QRS_NEXT_CUT()
PTP {E1 28256.982,E2 28256.982}
PTP {X 0,Y 607.876,A -85,B 0,C 180,E1 28256.982,E2 28256.982,E3 0,E4 0,E5 0,E6 0}
QRS_SPEED_INIT()
LIN {X 0,Y 607.876,Z 951,A -85,B 0,C 180,E1 28256.982,E2 28256.982,E3 0,E4 0,E5 0,E6 0} C_VEL
LIN {X 0,Y 607.876,Z 233.398,A -85,B 0,C 180,E1 28256.982,E2 28256.982} C_VEL
LIN {X 0,Y 607.876,Z 225.322,A -85,B 0,C 180,E1 28256.982,E2 28256.982} C_VEL
LIN {X 0,Y 607.869,Z 223.322,A -85,B 0,C 180,E1 28256.793,E2 28256.793} C_VEL
LIN {X 0,Y 607.913,Z 223.325,A -85,B 0,C 180,E1 28253.769,E2 28253.769} C_VEL
LIN {X 0,Y 607.873,Z 223.321,A -85,B 0,C 180,E1 28250.629,E2 28250.629} C_VEL
LIN {X 0,Y 607.911,Z 223.323,A -85,B 0,C 180,E1 28247.558,E2 28247.558} C_VEL
LIN {X 0,Y 607.877,Z 223.322,A -85,B 0,C 180,E1 28244.449,E2 28244.449} C_VEL
LIN {X 0,Y 607.908,Z 223.321,A -85,B 0,C 180,E1 28241.331,E2 28241.331} C_VEL
LIN {X 0,Y 607.881,Z 223.322,A -85,B 0,C 180,E1 28238.28,E2 28238.28} C_VEL
LIN {X 0,Y 607.906,Z 223.322,A -85,B 0,C 180,E1 28235.203,E2 28235.203} C_VEL
LIN {X 0,Y 607.886,Z 223.323,A -85,B 0,C 180,E1 28232.039,E2 28232.039} C_VEL
LIN {X 0,Y 607.905,Z 223.32,A -85,B 0,C 180,E1 28228.906,E2 28228.906} C_VEL
LIN {X 0,Y 607.894,Z 223.324,A -85,B 0,C 180,E1 28225.771,E2 28225.771} C_VEL
LIN {X 0,Y 607.909,Z 223.317,A -85,B 0,C 180,E1 28222.516,E2 28222.516} C_VEL
LIN {X 0,Y 607.913,Z 223.326,A -85,B 0,C 180,E1 28219.236,E2 28219.236} C_VEL
LIN {X 0,Y 607.898,Z 223.319,A -85,B 0,C 180,E1 28215.954,E2 28215.954} C_VEL
LIN {X 0,Y 607.896,Z 223.322,A -85,B 0,C 180,E1 28212.789,E2 28212.789} C_VEL
LIN {X 0,Y 607.898,Z 223.321,A -85,B 0,C 180,E1 28209.656,E2 28209.656} C_VEL
LIN {X 0,Y 607.891,Z 223.321,A -85,B 0,C 180,E1 28206.543,E2 28206.543} C_VEL
LIN {X 0,Y 607.902,Z 223.322,A -85,B 0,C 180,E1 28203.436,E2 28203.436} C_VEL
LIN {X 0,Y 607.889,Z 223.32,A -85,B 0,C 180,E1 28200.287,E2 28200.287} C_VEL
LIN {X 0,Y 607.91,Z 223.325,A -85,B 0,C 180,E1 28197.104,E2 28197.104} C_VEL
LIN {X 0,Y 607.899,Z 223.318,A -85,B 0,C 180,E1 28193.868,E2 28193.868} C_VEL
LIN {X 0,Y 607.897,Z 223.326,A -85,B 0,C 180,E1 28190.609,E2 28190.609} C_VEL
LIN {X 0,Y 607.916,Z 223.317,A -85,B 0,C 180,E1 28187.419,E2 28187.419} C_VEL
LIN {X 0,Y 607.881,Z 223.324,A -85,B 0,C 180,E1 28184.285,E2 28184.285} C_VEL
LIN {X 0,Y 607.914,Z 223.318,A -85,B 0,C 180,E1 28181.192,E2 28181.192} C_VEL
LIN {X 0,Y 607.873,Z 223.326,A -85,B 0,C 180,E1 28178.035,E2 28178.035} C_VEL
LIN {X 0,Y 607.913,Z 223.532,A -85,B 0,C 180,E1 28176.802,E2 28176.802} C_VEL
LIN {X 0,Y 607.916,Z 225.924,A -85,B 0,C 180,E1 28176.612,E2 28176.612} C_VEL
LIN {X 0,Y 607.89,Z 279.402,A -85,B 0,C 180,E1 28173.632,E2 28173.632} C_VEL
LIN {X 0,Y 607.913,Z 336.91,A -85,B 0,C 180,E1 28170.519,E2 28170.519} C_VEL
LIN {X 0,Y 607.902,Z 395.097,A -85,B 0,C 180,E1 28167.456,E2 28167.456} C_VEL
LIN {X 0,Y 607.896,Z 417.723,A -85,B 0,C 180,E1 28166.3,E2 28166.3} C_VEL
LIN {X 0,Y 607.917,Z 627.491,A -85,B 0,C 180,E1 28163.674,E2 28163.674} C_VEL
LIN {X 0,Y 607.913,Z 646.173,A -85,B 0,C 180,E1 28163.271,E2 28163.271} C_VEL
LIN {X 0,Y 607.918,Z 664.898,A -85,B 0,C 180,E1 28162.681,E2 28162.681} C_VEL
LIN {X 0,Y 607.911,Z 682.608,A -85,B 0,C 180,E1 28161.94,E2 28161.94} C_VEL
LIN {X 0,Y 607.919,Z 700.049,A -85,B 0,C 180,E1 28161.012,E2 28161.012} C_VEL
LIN {X 0,Y 607.919,Z 716.108,A -85,B 0,C 180,E1 28159.961,E2 28159.961} C_VEL
LIN {X 0,Y 607.915,Z 731.242,A -85,B 0,C 180,E1 28158.762,E2 28158.762} C_VEL
LIN {X 0,Y 607.916,Z 744.939,A -85,B 0,C 180,E1 28157.462,E2 28157.462} C_VEL
LIN {X 0,Y 607.919,Z 757.696,A -85,B 0,C 180,E1 28156.01,E2 28156.01} C_VEL
LIN {X 0,Y 607.915,Z 769.022,A -85,B 0,C 180,E1 28154.45,E2 28154.45} C_VEL
LIN {X 0,Y 607.913,Z 778.456,A -85,B 0,C 180,E1 28152.858,E2 28152.858} C_VEL
LIN {X 0,Y 607.908,Z 786.332,A -85,B 0,C 180,E1 28151.195,E2 28151.195} C_VEL
LIN {X 0,Y 607.913,Z 792.505,A -85,B 0,C 180,E1 28149.494,E2 28149.494} C_VEL
LIN {X 0,Y 607.919,Z 796.976,A -85,B 0,C 180,E1 28147.774,E2 28147.774} C_VEL
LIN {X 0,Y 607.908,Z 799.783,A -85,B 0,C 180,E1 28146.032,E2 28146.032} C_VEL
LIN {X 0,Y 607.912,Z 800.933,A -85,B 0,C 180,E1 28144.266,E2 28144.266} C_VEL
LIN {X 0,Y 607.912,Z 800.367,A -85,B 0,C 180,E1 28142.474,E2 28142.474} C_VEL
LIN {X 0,Y 607.912,Z 798.18,A -85,B 0,C 180,E1 28140.76,E2 28140.76} C_VEL
LIN {X 0,Y 607.914,Z 794.265,A -85,B 0,C 180,E1 28139.017,E2 28139.017} C_VEL
LIN {X 0,Y 607.908,Z 788.856,A -85,B 0,C 180,E1 28137.353,E2 28137.353} C_VEL
LIN {X 0,Y 607.916,Z 781.522,A -85,B 0,C 180,E1 28135.654,E2 28135.654} C_VEL
LIN {X 0,Y 607.913,Z 772.553,A -85,B 0,C 180,E1 28134.018,E2 28134.018} C_VEL
LIN {X 0,Y 607.914,Z 762.445,A -85,B 0,C 180,E1 28132.517,E2 28132.517} C_VEL
LIN {X 0,Y 607.915,Z 750.725,A -85,B 0,C 180,E1 28131.073,E2 28131.073} C_VEL
LIN {X 0,Y 607.914,Z 737.718,A -85,B 0,C 180,E1 28129.733,E2 28129.733} C_VEL
LIN {X 0,Y 607.917,Z 723.253,A -85,B 0,C 180,E1 28128.486,E2 28128.486} C_VEL
LIN {X 0,Y 607.917,Z 707.272,A -85,B 0,C 180,E1 28127.343,E2 28127.343} C_VEL
LIN {X 0,Y 607.896,Z 690.448,A -85,B 0,C 180,E1 28126.36,E2 28126.36} C_VEL
LIN {X 0,Y 607.915,Z 672.447,A -85,B 0,C 180,E1 28125.522,E2 28125.522} C_VEL
LIN {X 0,Y 607.915,Z 654.423,A -85,B 0,C 180,E1 28124.876,E2 28124.876} C_VEL
LIN {X 0,Y 607.913,Z 636.158,A -85,B 0,C 180,E1 28124.401,E2 28124.401} C_VEL
LIN {X 0,Y 607.919,Z 616.8,A -85,B 0,C 180,E1 28124.083,E2 28124.083} C_VEL
LIN {X 0,Y 607.917,Z 417.224,A -85,B 0,C 180,E1 28121.598,E2 28121.598} C_VEL
LIN {X 0,Y 607.897,Z 358.995,A -85,B 0,C 180,E1 28118.562,E2 28118.562} C_VEL
LIN {X 0,Y 607.915,Z 298.763,A -85,B 0,C 180,E1 28115.337,E2 28115.337} C_VEL
LIN {X 0,Y 607.915,Z 242.721,A -85,B 0,C 180,E1 28112.245,E2 28112.245} C_VEL
LIN {X 0,Y 607.894,Z 223.784,A -85,B 0,C 180,E1 28111.15,E2 28111.15} C_VEL
LIN {X 0,Y 607.854,Z 223.332,A -85,B 0,C 180,E1 28110.839,E2 28110.839} C_VEL
LIN {X 0,Y 607.831,Z 223.328,A -85,B 0,C 180,E1 28108.063,E2 28108.063} C_VEL
LIN {X 0,Y 607.896,Z 223.327,A -85,B 0,C 180,E1 28105.005,E2 28105.005} C_VEL
LIN {X 0,Y 607.827,Z 223.327,A -85,B 0,C 180,E1 28102.129,E2 28102.129} C_VEL
LIN {X 0,Y 607.89,Z 223.327,A -85,B 0,C 180,E1 28099.205,E2 28099.205} C_VEL
LIN {X 0,Y 607.83,Z 223.327,A -85,B 0,C 180,E1 28096.131,E2 28096.131} C_VEL
LIN {X 0,Y 607.845,Z 223.327,A -85,B 0,C 180,E1 28093.41,E2 28093.41} C_VEL
LIN {X 0,Y 607.839,Z 223.327,A -85,B 0,C 180,E1 28090.137,E2 28090.137} C_VEL
LIN {X 0,Y 607.83,Z 223.327,A -85,B 0,C 180,E1 28087.466,E2 28087.466} C_VEL
LIN {X 0,Y 607.877,Z 223.327,A -85,B 0,C 180,E1 28084.339,E2 28084.339} C_VEL
LIN {X 0,Y 607.824,Z 223.327,A -85,B 0,C 180,E1 28081.508,E2 28081.508} C_VEL
LIN {X 0,Y 607.913,Z 223.327,A -85,B 0,C 180,E1 28078.492,E2 28078.492} C_VEL
LIN {X 0,Y 607.824,Z 223.327,A -85,B 0,C 180,E1 28075.471,E2 28075.471} C_VEL
LIN {X 0,Y 607.845,Z 223.327,A -85,B 0,C 180,E1 28072.818,E2 28072.818} C_VEL
LIN {X 0,Y 607.836,Z 223.328,A -85,B 0,C 180,E1 28069.575,E2 28069.575} C_VEL
LIN {X 0,Y 607.83,Z 223.327,A -85,B 0,C 180,E1 28066.853,E2 28066.853} C_VEL
LIN {X 0,Y 607.859,Z 223.327,A -85,B 0,C 180,E1 28063.663,E2 28063.663} C_VEL
LIN {X 0,Y 607.823,Z 223.327,A -85,B 0,C 180,E1 28060.892,E2 28060.892} C_VEL
LIN {X 0,Y 607.905,Z 223.327,A -85,B 0,C 180,E1 28057.815,E2 28057.815} C_VEL
LIN {X 0,Y 607.824,Z 223.327,A -85,B 0,C 180,E1 28054.887,E2 28054.887} C_VEL
LIN {X 0,Y 607.871,Z 223.328,A -85,B 0,C 180,E1 28052.038,E2 28052.038} C_VEL
LIN {X 0,Y 607.83,Z 223.327,A -85,B 0,C 180,E1 28048.901,E2 28048.901} C_VEL
LIN {X 0,Y 607.837,Z 223.327,A -85,B 0,C 180,E1 28046.221,E2 28046.221} C_VEL
LIN {X 0,Y 607.839,Z 223.327,A -85,B 0,C 180,E1 28042.865,E2 28042.865} C_VEL
LIN {X 0,Y 607.835,Z 223.328,A -85,B 0,C 180,E1 28040.094,E2 28040.094} C_VEL
LIN {X 0,Y 607.86,Z 223.326,A -85,B 0,C 180,E1 28036.912,E2 28036.912} C_VEL
LIN {X 0,Y 607.829,Z 223.327,A -85,B 0,C 180,E1 28034.091,E2 28034.091} C_VEL
LIN {X 0,Y 607.873,Z 223.59,A -85,B 0,C 180,E1 28031.49,E2 28031.49} C_VEL
LIN {X 0,Y 607.887,Z 224.472,A -85,B 0,C 180,E1 28031.391,E2 28031.391} C_VEL
LIN {X 0,Y 607.917,Z 283.251,A -85,B 0,C 180,E1 28028.68,E2 28028.68} C_VEL
LIN {X 0,Y 607.918,Z 312.017,A -85,B 0,C 180,E1 28027.401,E2 28027.401} C_VEL
LIN {X 0,Y 607.918,Z 518.654,A -85,B 0,C 180,E1 28024.442,E2 28024.442} C_VEL
LIN {X 0,Y 607.912,Z 661.034,A -85,B 0,C 180,E1 28022.442,E2 28022.442} C_VEL
LIN {X 0,Y 607.919,Z 684.142,A -85,B 0,C 180,E1 28021.955,E2 28021.955} C_VEL
LIN {X 0,Y 607.916,Z 703.574,A -85,B 0,C 180,E1 28021.393,E2 28021.393} C_VEL
LIN {X 0,Y 607.913,Z 724.964,A -85,B 0,C 180,E1 28020.626,E2 28020.626} C_VEL
LIN {X 0,Y 607.919,Z 745.116,A -85,B 0,C 180,E1 28019.725,E2 28019.725} C_VEL
LIN {X 0,Y 607.916,Z 765.788,A -85,B 0,C 180,E1 28018.647,E2 28018.647} C_VEL
LIN {X 0,Y 607.917,Z 785.585,A -85,B 0,C 180,E1 28017.419,E2 28017.419} C_VEL
LIN {X 0,Y 607.915,Z 804.976,A -85,B 0,C 180,E1 28016.048,E2 28016.048} C_VEL
LIN {X 0,Y 607.912,Z 823.181,A -85,B 0,C 180,E1 28014.558,E2 28014.558} C_VEL
LIN {X 0,Y 607.909,Z 841.611,A -85,B 0,C 180,E1 28012.839,E2 28012.839} C_VEL
LIN {X 0,Y 607.905,Z 857.887,A -85,B 0,C 180,E1 28011.111,E2 28011.111} C_VEL
LIN {X 0,Y 607.906,Z 873.086,A -85,B 0,C 180,E1 28009.25,E2 28009.25} C_VEL
LIN {X 0,Y 607.907,Z 887.525,A -85,B 0,C 180,E1 28007.22,E2 28007.22} C_VEL
LIN {X 0,Y 607.916,Z 899.042,A -85,B 0,C 180,E1 28005.354,E2 28005.354} C_VEL
LIN {X 0,Y 607.917,Z 909.76,A -85,B 0,C 180,E1 28003.311,E2 28003.311} C_VEL
LIN {X 0,Y 607.916,Z 918.789,A -85,B 0,C 180,E1 28001.286,E2 28001.286} C_VEL
LIN {X 0,Y 607.919,Z 926.346,A -85,B 0,C 180,E1 27999.179,E2 27999.179} C_VEL
LIN {X 0,Y 607.913,Z 932.358,A -85,B 0,C 180,E1 27997.085,E2 27997.085} C_VEL
LIN {X 0,Y 607.908,Z 936.64,A -85,B 0,C 180,E1 27995,E2 27995} C_VEL
LIN {X 0,Y 607.915,Z 939.406,A -85,B 0,C 180,E1 27993.016,E2 27993.016} C_VEL
LIN {X 0,Y 607.906,Z 940.806,A -85,B 0,C 180,E1 27990.847,E2 27990.847} C_VEL
LIN {X 0,Y 607.918,Z 940.738,A -85,B 0,C 180,E1 27988.868,E2 27988.868} C_VEL
LIN {X 0,Y 607.909,Z 939.065,A -85,B 0,C 180,E1 27986.699,E2 27986.699} C_VEL
LIN {X 0,Y 607.909,Z 936.159,A -85,B 0,C 180,E1 27984.714,E2 27984.714} C_VEL
LIN {X 0,Y 607.913,Z 931.332,A -85,B 0,C 180,E1 27982.533,E2 27982.533} C_VEL
LIN {X 0,Y 607.91,Z 925.729,A -85,B 0,C 180,E1 27980.628,E2 27980.628} C_VEL
LIN {X 0,Y 607.91,Z 917.553,A -85,B 0,C 180,E1 27978.424,E2 27978.424} C_VEL
LIN {X 0,Y 607.918,Z 909.286,A -85,B 0,C 180,E1 27976.59,E2 27976.59} C_VEL
LIN {X 0,Y 607.912,Z 897.869,A -85,B 0,C 180,E1 27974.448,E2 27974.448} C_VEL
LIN {X 0,Y 607.919,Z 886.225,A -85,B 0,C 180,E1 27972.581,E2 27972.581} C_VEL
LIN {X 0,Y 607.915,Z 871.875,A -85,B 0,C 180,E1 27970.595,E2 27970.595} C_VEL
LIN {X 0,Y 607.91,Z 856.976,A -85,B 0,C 180,E1 27968.786,E2 27968.786} C_VEL
LIN {X 0,Y 607.909,Z 840.575,A -85,B 0,C 180,E1 27967.057,E2 27967.057} C_VEL
LIN {X 0,Y 607.917,Z 822.199,A -85,B 0,C 180,E1 27965.358,E2 27965.358} C_VEL
LIN {X 0,Y 607.914,Z 803.588,A -85,B 0,C 180,E1 27963.845,E2 27963.845} C_VEL
LIN {X 0,Y 607.918,Z 784.749,A -85,B 0,C 180,E1 27962.525,E2 27962.525} C_VEL
LIN {X 0,Y 607.917,Z 764.763,A -85,B 0,C 180,E1 27961.297,E2 27961.297} C_VEL
LIN {X 0,Y 607.919,Z 745.116,A -85,B 0,C 180,E1 27960.275,E2 27960.275} C_VEL
LIN {X 0,Y 607.914,Z 724.087,A -85,B 0,C 180,E1 27959.339,E2 27959.339} C_VEL
LIN {X 0,Y 607.916,Z 703.574,A -85,B 0,C 180,E1 27958.607,E2 27958.607} C_VEL
LIN {X 0,Y 607.919,Z 684.1,A -85,B 0,C 180,E1 27958.044,E2 27958.044} C_VEL
LIN {X 0,Y 607.911,Z 662.086,A -85,B 0,C 180,E1 27957.575,E2 27957.575} C_VEL
LIN {X 0,Y 607.908,Z 431.434,A -85,B 0,C 180,E1 27954.325,E2 27954.325} C_VEL
LIN {X 0,Y 607.918,Z 311.433,A -85,B 0,C 180,E1 27952.578,E2 27952.578} C_VEL
LIN {X 0,Y 607.918,Z 247.749,A -85,B 0,C 180,E1 27949.699,E2 27949.699} C_VEL
LIN {X 0,Y 607.88,Z 223.942,A -85,B 0,C 180,E1 27948.565,E2 27948.565} C_VEL
LIN {X 0,Y 607.855,Z 223.344,A -85,B 0,C 180,E1 27948.352,E2 27948.352} C_VEL
LIN {X 0,Y 607.826,Z 223.327,A -85,B 0,C 180,E1 27945.643,E2 27945.643} C_VEL
LIN {X 0,Y 607.893,Z 223.327,A -85,B 0,C 180,E1 27942.533,E2 27942.533} C_VEL
LIN {X 0,Y 607.828,Z 223.327,A -85,B 0,C 180,E1 27939.659,E2 27939.659} C_VEL
LIN {X 0,Y 607.911,Z 223.328,A -85,B 0,C 180,E1 27936.617,E2 27936.617} C_VEL
LIN {X 0,Y 607.834,Z 223.326,A -85,B 0,C 180,E1 27933.553,E2 27933.553} C_VEL
LIN {X 0,Y 607.892,Z 223.327,A -85,B 0,C 180,E1 27930.656,E2 27930.656} C_VEL
LIN {X 0,Y 607.843,Z 223.325,A -85,B 0,C 180,E1 27927.531,E2 27927.531} C_VEL
LIN {X 0,Y 607.891,Z 223.327,A -85,B 0,C 180,E1 27924.591,E2 27924.591} C_VEL
LIN {X 0,Y 607.85,Z 223.324,A -85,B 0,C 180,E1 27921.418,E2 27921.418} C_VEL
LIN {X 0,Y 607.9,Z 223.327,A -85,B 0,C 180,E1 27918.409,E2 27918.409} C_VEL
LIN {X 0,Y 607.855,Z 223.323,A -85,B 0,C 180,E1 27915.259,E2 27915.259} C_VEL
LIN {X 0,Y 607.905,Z 223.328,A -85,B 0,C 180,E1 27912.25,E2 27912.25} C_VEL
LIN {X 0,Y 607.859,Z 223.323,A -85,B 0,C 180,E1 27909.086,E2 27909.086} C_VEL
LIN {X 0,Y 607.918,Z 223.326,A -85,B 0,C 180,E1 27906.043,E2 27906.043} C_VEL
LIN {X 0,Y 607.864,Z 223.323,A -85,B 0,C 180,E1 27902.923,E2 27902.923} C_VEL
LIN {X 0,Y 607.916,Z 223.326,A -85,B 0,C 180,E1 27899.906,E2 27899.906} C_VEL
LIN {X 0,Y 607.869,Z 223.322,A -85,B 0,C 180,E1 27896.793,E2 27896.793} C_VEL
LIN {X 0,Y 606.876,Z 223.455,A -85,B 0,C 180,E1 27896.067,E2 27896.067} C_VEL
LIN {X 0,Y 600.494,Z 224.252,A -85,B 0,C 180,E1 27894.03,E2 27894.03} C_VEL
LIN {X 0,Y 599.974,Z 224.31,A -85,B 0,C 180,E1 27893.5,E2 27893.5} C_VEL
LIN {X 0,Y 599.935,Z 224.311,A -85,B 0,C 180,E1 27890.407,E2 27890.407} C_VEL
LIN {X 0,Y 599.973,Z 224.307,A -85,B 0,C 180,E1 27887.195,E2 27887.195} C_VEL
LIN {X 0,Y 599.958,Z 224.314,A -85,B 0,C 180,E1 27883.94,E2 27883.94} C_VEL
LIN {X 0,Y 599.95,Z 224.307,A -85,B 0,C 180,E1 27880.611,E2 27880.611} C_VEL
LIN {X 0,Y 599.971,Z 224.313,A -85,B 0,C 180,E1 27877.406,E2 27877.406} C_VEL
LIN {X 0,Y 599.945,Z 224.31,A -85,B 0,C 180,E1 27874.217,E2 27874.217} C_VEL
LIN {X 0,Y 599.966,Z 224.308,A -85,B 0,C 180,E1 27871.037,E2 27871.037} C_VEL
LIN {X 0,Y 599.953,Z 224.313,A -85,B 0,C 180,E1 27867.846,E2 27867.846} C_VEL
LIN {X 0,Y 599.97,Z 224.306,A -85,B 0,C 180,E1 27864.581,E2 27864.581} C_VEL
LIN {X 0,Y 599.973,Z 224.314,A -85,B 0,C 180,E1 27861.254,E2 27861.254} C_VEL
LIN {X 0,Y 599.959,Z 224.308,A -85,B 0,C 180,E1 27858.012,E2 27858.012} C_VEL
LIN {X 0,Y 599.958,Z 224.311,A -85,B 0,C 180,E1 27854.826,E2 27854.826} C_VEL
LIN {X 0,Y 599.959,Z 224.31,A -85,B 0,C 180,E1 27851.679,E2 27851.679} C_VEL
LIN {X 0,Y 599.954,Z 224.31,A -85,B 0,C 180,E1 27848.558,E2 27848.558} C_VEL
LIN {X 0,Y 599.964,Z 224.312,A -85,B 0,C 180,E1 27845.421,E2 27845.421} C_VEL
LIN {X 0,Y 599.955,Z 224.308,A -85,B 0,C 180,E1 27842.229,E2 27842.229} C_VEL
LIN {X 0,Y 599.971,Z 224.316,A -85,B 0,C 180,E1 27838.966,E2 27838.966} C_VEL
LIN {X 0,Y 599.976,Z 224.306,A -85,B 0,C 180,E1 27835.636,E2 27835.636} C_VEL
LIN {X 0,Y 599.945,Z 224.308,A -85,B 0,C 180,E1 27832.437,E2 27832.437} C_VEL
LIN {X 0,Y 599.97,Z 224.31,A -85,B 0,C 180,E1 27829.268,E2 27829.268} C_VEL
LIN {X 0,Y 599.939,Z 224.31,A -85,B 0,C 180,E1 27826.161,E2 27826.161} C_VEL
LIN {X 0,Y 599.971,Z 224.312,A -85,B 0,C 180,E1 27823.002,E2 27823.002} C_VEL
LIN {X 0,Y 599.935,Z 224.312,A -85,B 0,C 180,E1 27819.885,E2 27819.885} C_VEL
LIN {X 0,Y 599.992,Z 224.477,A -85,B 0,C 180,E1 27817.277,E2 27817.277} C_VEL
LIN {X 0,Y 600.467,Z 226.248,A -85,B 0,C 180,E1 27817.066,E2 27817.066} C_VEL
LIN {X 0,Y 600.943,Z 227.973,A -85,B 0,C 180,E1 27816.929,E2 27816.929} C_VEL
LIN {X 0,Y 600.723,Z 280.481,A -85,B 0,C 180,E1 27813.962,E2 27813.962} C_VEL
LIN {X 0,Y 600.585,Z 337.974,A -85,B 0,C 180,E1 27810.812,E2 27810.812} C_VEL
LIN {X 0,Y 600.431,Z 396.149,A -85,B 0,C 180,E1 27807.711,E2 27807.711} C_VEL
LIN {X 0,Y 600.462,Z 418.081,A -85,B 0,C 180,E1 27806.585,E2 27806.585} C_VEL
LIN {X 0,Y 600.377,Z 628.417,A -85,B 0,C 180,E1 27803.916,E2 27803.916} C_VEL
LIN {X 0,Y 600.334,Z 647.321,A -85,B 0,C 180,E1 27803.492,E2 27803.492} C_VEL
LIN {X 0,Y 600.295,Z 665.08,A -85,B 0,C 180,E1 27802.921,E2 27802.921} C_VEL
LIN {X 0,Y 600.227,Z 683.158,A -85,B 0,C 180,E1 27802.15,E2 27802.15} C_VEL
LIN {X 0,Y 600.177,Z 700.139,A -85,B 0,C 180,E1 27801.233,E2 27801.233} C_VEL
LIN {X 0,Y 600.119,Z 716.195,A -85,B 0,C 180,E1 27800.168,E2 27800.168} C_VEL
LIN {X 0,Y 600.064,Z 731.534,A -85,B 0,C 180,E1 27798.934,E2 27798.934} C_VEL
LIN {X 0,Y 600.018,Z 745.821,A -85,B 0,C 180,E1 27797.55,E2 27797.55} C_VEL
LIN {X 0,Y 599.984,Z 758.138,A -85,B 0,C 180,E1 27796.116,E2 27796.116} C_VEL
LIN {X 0,Y 599.953,Z 768.734,A -85,B 0,C 180,E1 27794.635,E2 27794.635} C_VEL
LIN {X 0,Y 599.934,Z 778.102,A -85,B 0,C 180,E1 27793.044,E2 27793.044} C_VEL
LIN {X 0,Y 599.92,Z 786.135,A -85,B 0,C 180,E1 27791.339,E2 27791.339} C_VEL
LIN {X 0,Y 599.915,Z 792.355,A -85,B 0,C 180,E1 27789.616,E2 27789.616} C_VEL
LIN {X 0,Y 599.915,Z 796.872,A -85,B 0,C 180,E1 27787.874,E2 27787.874} C_VEL
LIN {X 0,Y 599.911,Z 799.725,A -85,B 0,C 180,E1 27786.11,E2 27786.11} C_VEL
LIN {X 0,Y 599.913,Z 800.921,A -85,B 0,C 180,E1 27784.322,E2 27784.322} C_VEL
LIN {X 0,Y 599.912,Z 800.404,A -85,B 0,C 180,E1 27782.507,E2 27782.507} C_VEL
LIN {X 0,Y 599.913,Z 798.267,A -85,B 0,C 180,E1 27780.77,E2 27780.77} C_VEL
LIN {X 0,Y 599.916,Z 794.405,A -85,B 0,C 180,E1 27779.004,E2 27779.004} C_VEL
LIN {X 0,Y 599.915,Z 789.04,A -85,B 0,C 180,E1 27777.315,E2 27777.315} C_VEL
LIN {X 0,Y 599.93,Z 781.726,A -85,B 0,C 180,E1 27775.585,E2 27775.585} C_VEL
LIN {X 0,Y 599.944,Z 772.815,A -85,B 0,C 180,E1 27773.928,E2 27773.928} C_VEL
LIN {X 0,Y 599.967,Z 762.233,A -85,B 0,C 180,E1 27772.334,E2 27772.334} C_VEL
LIN {X 0,Y 600.005,Z 750.168,A -85,B 0,C 180,E1 27770.836,E2 27770.836} C_VEL
LIN {X 0,Y 600.046,Z 736.755,A -85,B 0,C 180,E1 27769.448,E2 27769.448} C_VEL
LIN {X 0,Y 600.1,Z 722.366,A -85,B 0,C 180,E1 27768.207,E2 27768.207} C_VEL
LIN {X 0,Y 600.165,Z 706.154,A -85,B 0,C 180,E1 27767.05,E2 27767.05} C_VEL
LIN {X 0,Y 600.201,Z 689.246,A -85,B 0,C 180,E1 27766.066,E2 27766.066} C_VEL
LIN {X 0,Y 600.277,Z 671.472,A -85,B 0,C 180,E1 27765.241,E2 27765.241} C_VEL
LIN {X 0,Y 600.329,Z 653.421,A -85,B 0,C 180,E1 27764.596,E2 27764.596} C_VEL
LIN {X 0,Y 600.365,Z 635.055,A -85,B 0,C 180,E1 27764.124,E2 27764.124} C_VEL
LIN {X 0,Y 600.396,Z 615.218,A -85,B 0,C 180,E1 27763.804,E2 27763.804} C_VEL
LIN {X 0,Y 600.414,Z 417.383,A -85,B 0,C 180,E1 27761.309,E2 27761.309} C_VEL
LIN {X 0,Y 600.51,Z 359.145,A -85,B 0,C 180,E1 27758.235,E2 27758.235} C_VEL
LIN {X 0,Y 600.695,Z 298.206,A -85,B 0,C 180,E1 27754.93,E2 27754.93} C_VEL
LIN {X 0,Y 600.865,Z 242.853,A -85,B 0,C 180,E1 27751.836,E2 27751.836} C_VEL
LIN {X 0,Y 600.957,Z 227.382,A -85,B 0,C 180,E1 27750.937,E2 27750.937} C_VEL
LIN {X 0,Y 599.956,Z 224.693,A -85,B 0,C 180,E1 27750.661,E2 27750.661} C_VEL
LIN {X 0,Y 599.898,Z 224.316,A -85,B 0,C 180,E1 27750,E2 27750} C_VEL
LIN {X 0,Y 599.916,Z 224.318,A -85,B 0,C 180,E1 27746.743,E2 27746.743} C_VEL
LIN {X 0,Y 599.891,Z 224.315,A -85,B 0,C 180,E1 27743.996,E2 27743.996} C_VEL
LIN {X 0,Y 599.956,Z 224.317,A -85,B 0,C 180,E1 27740.894,E2 27740.894} C_VEL
LIN {X 0,Y 599.889,Z 224.316,A -85,B 0,C 180,E1 27737.884,E2 27737.884} C_VEL
LIN {X 0,Y 599.963,Z 224.317,A -85,B 0,C 180,E1 27734.772,E2 27734.772} C_VEL
LIN {X 0,Y 599.887,Z 224.316,A -85,B 0,C 180,E1 27731.732,E2 27731.732} C_VEL
LIN {X 0,Y 599.962,Z 224.316,A -85,B 0,C 180,E1 27728.626,E2 27728.626} C_VEL
LIN {X 0,Y 599.886,Z 224.316,A -85,B 0,C 180,E1 27725.643,E2 27725.643} C_VEL
LIN {X 0,Y 599.96,Z 224.316,A -85,B 0,C 180,E1 27722.674,E2 27722.674} C_VEL
LIN {X 0,Y 599.887,Z 224.316,A -85,B 0,C 180,E1 27719.618,E2 27719.618} C_VEL
LIN {X 0,Y 599.915,Z 224.316,A -85,B 0,C 180,E1 27716.847,E2 27716.847} C_VEL
LIN {X 0,Y 599.897,Z 224.316,A -85,B 0,C 180,E1 27713.684,E2 27713.684} C_VEL
LIN {X 0,Y 599.89,Z 224.316,A -85,B 0,C 180,E1 27710.986,E2 27710.986} C_VEL
LIN {X 0,Y 599.921,Z 224.317,A -85,B 0,C 180,E1 27707.78,E2 27707.78} C_VEL
LIN {X 0,Y 599.886,Z 224.316,A -85,B 0,C 180,E1 27704.929,E2 27704.929} C_VEL
LIN {X 0,Y 599.952,Z 224.317,A -85,B 0,C 180,E1 27701.841,E2 27701.841} C_VEL
LIN {X 0,Y 599.884,Z 224.316,A -85,B 0,C 180,E1 27698.899,E2 27698.899} C_VEL
LIN {X 0,Y 599.967,Z 224.316,A -85,B 0,C 180,E1 27695.902,E2 27695.902} C_VEL
LIN {X 0,Y 599.886,Z 224.317,A -85,B 0,C 180,E1 27692.826,E2 27692.826} C_VEL
LIN {X 0,Y 599.948,Z 224.317,A -85,B 0,C 180,E1 27689.874,E2 27689.874} C_VEL
LIN {X 0,Y 599.888,Z 224.317,A -85,B 0,C 180,E1 27686.746,E2 27686.746} C_VEL
LIN {X 0,Y 599.94,Z 224.317,A -85,B 0,C 180,E1 27683.766,E2 27683.766} C_VEL
LIN {X 0,Y 599.892,Z 224.317,A -85,B 0,C 180,E1 27680.654,E2 27680.654} C_VEL
LIN {X 0,Y 599.909,Z 224.318,A -85,B 0,C 180,E1 27677.872,E2 27677.872} C_VEL
LIN {X 0,Y 599.901,Z 224.316,A -85,B 0,C 180,E1 27674.628,E2 27674.628} C_VEL
LIN {X 0,Y 599.919,Z 224.53,A -85,B 0,C 180,E1 27672.127,E2 27672.127} C_VEL
LIN {X 0,Y 600.303,Z 226.02,A -85,B 0,C 180,E1 27671.954,E2 27671.954} C_VEL
LIN {X 0,Y 601.629,Z 228.601,A -85,B 0,C 180,E1 27671.717,E2 27671.717} C_VEL
LIN {X 0,Y 601.429,Z 290.607,A -85,B 0,C 180,E1 27668.84,E2 27668.84} C_VEL
LIN {X 0,Y 601.508,Z 313.14,A -85,B 0,C 180,E1 27667.846,E2 27667.846} C_VEL
LIN {X 0,Y 601.315,Z 517.805,A -85,B 0,C 180,E1 27664.886,E2 27664.886} C_VEL
LIN {X 0,Y 601.146,Z 662.228,A -85,B 0,C 180,E1 27662.833,E2 27662.833} C_VEL
LIN {X 0,Y 601.072,Z 685.852,A -85,B 0,C 180,E1 27662.316,E2 27662.316} C_VEL
LIN {X 0,Y 601,Z 705.268,A -85,B 0,C 180,E1 27661.741,E2 27661.741} C_VEL
LIN {X 0,Y 600.878,Z 727.589,A -85,B 0,C 180,E1 27660.91,E2 27660.91} C_VEL
LIN {X 0,Y 600.793,Z 747.333,A -85,B 0,C 180,E1 27660.005,E2 27660.005} C_VEL
LIN {X 0,Y 600.656,Z 768.494,A -85,B 0,C 180,E1 27658.863,E2 27658.863} C_VEL
LIN {X 0,Y 600.556,Z 787.915,A -85,B 0,C 180,E1 27657.628,E2 27657.628} C_VEL
LIN {X 0,Y 600.423,Z 807.946,A -85,B 0,C 180,E1 27656.159,E2 27656.159} C_VEL
LIN {X 0,Y 600.326,Z 826.727,A -85,B 0,C 180,E1 27654.581,E2 27654.581} C_VEL
LIN {X 0,Y 600.224,Z 844.044,A -85,B 0,C 180,E1 27652.899,E2 27652.899} C_VEL
LIN {X 0,Y 600.12,Z 861.295,A -85,B 0,C 180,E1 27650.989,E2 27650.989} C_VEL
LIN {X 0,Y 600.058,Z 876.002,A -85,B 0,C 180,E1 27649.131,E2 27649.131} C_VEL
LIN {X 0,Y 600.009,Z 888.812,A -85,B 0,C 180,E1 27647.253,E2 27647.253} C_VEL
LIN {X 0,Y 599.976,Z 900.922,A -85,B 0,C 180,E1 27645.226,E2 27645.226} C_VEL
LIN {X 0,Y 599.951,Z 910.775,A -85,B 0,C 180,E1 27643.277,E2 27643.277} C_VEL
LIN {X 0,Y 599.923,Z 919.915,A -85,B 0,C 180,E1 27641.146,E2 27641.146} C_VEL
LIN {X 0,Y 599.927,Z 926.956,A -85,B 0,C 180,E1 27639.109,E2 27639.109} C_VEL
LIN {X 0,Y 599.91,Z 933.016,A -85,B 0,C 180,E1 27636.891,E2 27636.891} C_VEL
LIN {X 0,Y 599.901,Z 936.959,A -85,B 0,C 180,E1 27634.875,E2 27634.875} C_VEL
LIN {X 0,Y 599.916,Z 939.786,A -85,B 0,C 180,E1 27632.674,E2 27632.674} C_VEL
LIN {X 0,Y 599.896,Z 940.873,A -85,B 0,C 180,E1 27630.572,E2 27630.572} C_VEL
LIN {X 0,Y 599.896,Z 940.524,A -85,B 0,C 180,E1 27628.375,E2 27628.375} C_VEL
LIN {X 0,Y 599.908,Z 938.727,A -85,B 0,C 180,E1 27626.368,E2 27626.368} C_VEL
LIN {X 0,Y 599.9,Z 935.285,A -85,B 0,C 180,E1 27624.164,E2 27624.164} C_VEL
LIN {X 0,Y 599.912,Z 930.567,A -85,B 0,C 180,E1 27622.144,E2 27622.144} C_VEL
LIN {X 0,Y 599.912,Z 924.18,A -85,B 0,C 180,E1 27620.017,E2 27620.017} C_VEL
LIN {X 0,Y 599.923,Z 916.327,A -85,B 0,C 180,E1 27617.975,E2 27617.975} C_VEL
LIN {X 0,Y 599.96,Z 906.924,A -85,B 0,C 180,E1 27615.912,E2 27615.912} C_VEL
LIN {X 0,Y 599.984,Z 896.129,A -85,B 0,C 180,E1 27613.94,E2 27613.94} C_VEL
LIN {X 0,Y 600.03,Z 883.574,A -85,B 0,C 180,E1 27611.944,E2 27611.944} C_VEL
LIN {X 0,Y 600.082,Z 870.32,A -85,B 0,C 180,E1 27610.128,E2 27610.128} C_VEL
LIN {X 0,Y 600.173,Z 854.188,A -85,B 0,C 180,E1 27608.191,E2 27608.191} C_VEL
LIN {X 0,Y 600.268,Z 837.523,A -85,B 0,C 180,E1 27606.436,E2 27606.436} C_VEL
LIN {X 0,Y 600.345,Z 819.784,A -85,B 0,C 180,E1 27604.815,E2 27604.815} C_VEL
LIN {X 0,Y 600.481,Z 799.387,A -85,B 0,C 180,E1 27603.188,E2 27603.188} C_VEL
LIN {X 0,Y 600.601,Z 779.925,A -85,B 0,C 180,E1 27601.838,E2 27601.838} C_VEL
LIN {X 0,Y 600.716,Z 759.798,A -85,B 0,C 180,E1 27600.647,E2 27600.647} C_VEL
LIN {X 0,Y 600.843,Z 738.73,A -85,B 0,C 180,E1 27599.575,E2 27599.575} C_VEL
LIN {X 0,Y 600.941,Z 717.641,A -85,B 0,C 180,E1 27598.699,E2 27598.699} C_VEL
LIN {X 0,Y 601.033,Z 696.369,A -85,B 0,C 180,E1 27597.971,E2 27597.971} C_VEL
LIN {X 0,Y 601.109,Z 674.401,A -85,B 0,C 180,E1 27597.41,E2 27597.41} C_VEL
LIN {X 0,Y 601.159,Z 654.596,A -85,B 0,C 180,E1 27597.041,E2 27597.041} C_VEL
LIN {X 0,Y 601.401,Z 435.379,A -85,B 0,C 180,E1 27593.936,E2 27593.936} C_VEL
LIN {X 0,Y 601.4,Z 312.109,A -85,B 0,C 180,E1 27592.125,E2 27592.125} C_VEL
LIN {X 0,Y 601.574,Z 248.418,A -85,B 0,C 180,E1 27589.216,E2 27589.216} C_VEL
LIN {X 0,Y 601.594,Z 228.311,A -85,B 0,C 180,E1 27588.266,E2 27588.266} C_VEL
LIN {X 0,Y 599.98,Z 224.87,A -85,B 0,C 180,E1 27587.938,E2 27587.938} C_VEL
LIN {X 0,Y 599.888,Z 224.293,A -85,B 0,C 180,E1 27587.672,E2 27587.672} C_VEL
LIN {X 0,Y 599.949,Z 224.316,A -85,B 0,C 180,E1 27584.558,E2 27584.558} C_VEL
LIN {X 0,Y 599.888,Z 224.316,A -85,B 0,C 180,E1 27581.55,E2 27581.55} C_VEL
LIN {X 0,Y 599.957,Z 224.315,A -85,B 0,C 180,E1 27578.435,E2 27578.435} C_VEL
LIN {X 0,Y 599.894,Z 224.316,A -85,B 0,C 180,E1 27575.452,E2 27575.452} C_VEL
LIN {X 0,Y 599.968,Z 224.314,A -85,B 0,C 180,E1 27572.335,E2 27572.335} C_VEL
LIN {X 0,Y 599.9,Z 224.315,A -85,B 0,C 180,E1 27569.341,E2 27569.341} C_VEL
LIN {X 0,Y 599.972,Z 224.312,A -85,B 0,C 180,E1 27566.208,E2 27566.208} C_VEL
LIN {X 0,Y 599.906,Z 224.315,A -85,B 0,C 180,E1 27563.163,E2 27563.163} C_VEL
LIN {X 0,Y 599.976,Z 224.312,A -85,B 0,C 180,E1 27560.078,E2 27560.078} C_VEL
LIN {X 0,Y 599.912,Z 224.314,A -85,B 0,C 180,E1 27557.058,E2 27557.058} C_VEL
LIN {X 0,Y 599.977,Z 224.312,A -85,B 0,C 180,E1 27553.984,E2 27553.984} C_VEL
LIN {X 0,Y 599.919,Z 224.313,A -85,B 0,C 180,E1 27550.856,E2 27550.856} C_VEL
LIN {X 0,Y 599.97,Z 224.309,A -85,B 0,C 180,E1 27547.662,E2 27547.662} C_VEL
LIN {X 0,Y 599.929,Z 224.313,A -85,B 0,C 180,E1 27544.589,E2 27544.589} C_VEL
LIN {X 0,Y 599.956,Z 224.307,A -85,B 0,C 180,E1 27541.337,E2 27541.337} C_VEL
LIN {X 0,Y 599.954,Z 224.315,A -85,B 0,C 180,E1 27538.186,E2 27538.186} C_VEL
LIN {X 0,Y 599.938,Z 224.31,A -85,B 0,C 180,E1 27534.933,E2 27534.933} C_VEL
LIN {X 0,Y 599.974,Z 224.31,A -85,B 0,C 180,E1 27533.5,E2 27533.5} C_VEL
LIN {X 0,Y 598.983,Z 224.432,A -85,B 0,C 180,E1 27532.765,E2 27532.765} C_VEL
LIN {X 0,Y 592.516,Z 225.235,A -85,B 0,C 180,E1 27530.701,E2 27530.701} C_VEL
LIN {X 0,Y 592.008,Z 225.301,A -85,B 0,C 180,E1 27530.164,E2 27530.164} C_VEL
LIN {X 0,Y 592.011,Z 225.296,A -85,B 0,C 180,E1 27526.821,E2 27526.821} C_VEL
LIN {X 0,Y 592.035,Z 225.303,A -85,B 0,C 180,E1 27523.592,E2 27523.592} C_VEL
LIN {X 0,Y 592.003,Z 225.297,A -85,B 0,C 180,E1 27520.361,E2 27520.361} C_VEL
LIN {X 0,Y 592.03,Z 225.299,A -85,B 0,C 180,E1 27517.239,E2 27517.239} C_VEL
LIN {X 0,Y 592.009,Z 225.3,A -85,B 0,C 180,E1 27514.061,E2 27514.061} C_VEL
LIN {X 0,Y 592.036,Z 225.293,A -85,B 0,C 180,E1 27510.786,E2 27510.786} C_VEL
LIN {X 0,Y 592.032,Z 225.305,A -85,B 0,C 180,E1 27507.431,E2 27507.431} C_VEL
LIN {X 0,Y 592.016,Z 225.297,A -85,B 0,C 180,E1 27504.124,E2 27504.124} C_VEL
LIN {X 0,Y 592.022,Z 225.298,A -85,B 0,C 180,E1 27500.954,E2 27500.954} C_VEL
LIN {X 0,Y 592.018,Z 225.3,A -85,B 0,C 180,E1 27497.765,E2 27497.765} C_VEL
LIN {X 0,Y 592.022,Z 225.297,A -85,B 0,C 180,E1 27494.545,E2 27494.545} C_VEL
LIN {X 0,Y 592.032,Z 225.303,A -85,B 0,C 180,E1 27491.277,E2 27491.277} C_VEL
LIN {X 0,Y 592.032,Z 225.295,A -85,B 0,C 180,E1 27487.934,E2 27487.934} C_VEL
LIN {X 0,Y 592.015,Z 225.301,A -85,B 0,C 180,E1 27484.666,E2 27484.666} C_VEL
LIN {X 0,Y 592.025,Z 225.3,A -85,B 0,C 180,E1 27481.458,E2 27481.458} C_VEL
LIN {X 0,Y 592.009,Z 225.3,A -85,B 0,C 180,E1 27478.333,E2 27478.333} C_VEL
LIN {X 0,Y 592.031,Z 225.301,A -85,B 0,C 180,E1 27475.148,E2 27475.148} C_VEL
LIN {X 0,Y 592.013,Z 225.29,A -85,B 0,C 180,E1 27471.917,E2 27471.917} C_VEL
LIN {X 0,Y 592.022,Z 225.302,A -85,B 0,C 180,E1 27468.615,E2 27468.615} C_VEL
LIN {X 0,Y 592.034,Z 225.295,A -85,B 0,C 180,E1 27465.352,E2 27465.352} C_VEL
LIN {X 0,Y 592,Z 225.296,A -85,B 0,C 180,E1 27462.189,E2 27462.189} C_VEL
LIN {X 0,Y 592.034,Z 225.293,A -85,B 0,C 180,E1 27459.037,E2 27459.037} C_VEL
LIN {X 0,Y 592.032,Z 225.555,A -85,B 0,C 180,E1 27457.766,E2 27457.766} C_VEL
LIN {X 0,Y 593.125,Z 228.482,A -85,B 0,C 180,E1 27457.459,E2 27457.459} C_VEL
LIN {X 0,Y 594.164,Z 231.481,A -85,B 0,C 180,E1 27457.203,E2 27457.203} C_VEL
LIN {X 0,Y 593.626,Z 275.543,A -85,B 0,C 180,E1 27454.638,E2 27454.638} C_VEL
LIN {X 0,Y 593.295,Z 334.628,A -85,B 0,C 180,E1 27451.353,E2 27451.353} C_VEL
LIN {X 0,Y 592.998,Z 393.572,A -85,B 0,C 180,E1 27448.165,E2 27448.165} C_VEL
LIN {X 0,Y 592.972,Z 418.108,A -85,B 0,C 180,E1 27446.887,E2 27446.887} C_VEL
LIN {X 0,Y 592.859,Z 627.519,A -85,B 0,C 180,E1 27444.196,E2 27444.196} C_VEL
LIN {X 0,Y 592.779,Z 646.68,A -85,B 0,C 180,E1 27443.77,E2 27443.77} C_VEL
LIN {X 0,Y 592.687,Z 665.165,A -85,B 0,C 180,E1 27443.171,E2 27443.171} C_VEL
LIN {X 0,Y 592.56,Z 683.245,A -85,B 0,C 180,E1 27442.389,E2 27442.389} C_VEL
LIN {X 0,Y 592.451,Z 700.223,A -85,B 0,C 180,E1 27441.46,E2 27441.46} C_VEL
LIN {X 0,Y 592.332,Z 716.275,A -85,B 0,C 180,E1 27440.381,E2 27440.381} C_VEL
LIN {X 0,Y 592.221,Z 731.392,A -85,B 0,C 180,E1 27439.151,E2 27439.151} C_VEL
LIN {X 0,Y 592.129,Z 745.063,A -85,B 0,C 180,E1 27437.816,E2 27437.816} C_VEL
LIN {X 0,Y 592.051,Z 757.8,A -85,B 0,C 180,E1 27436.325,E2 27436.325} C_VEL
LIN {X 0,Y 591.994,Z 769.098,A -85,B 0,C 180,E1 27434.725,E2 27434.725} C_VEL
LIN {X 0,Y 591.956,Z 778.396,A -85,B 0,C 180,E1 27433.112,E2 27433.112} C_VEL
LIN {X 0,Y 591.931,Z 786.364,A -85,B 0,C 180,E1 27431.384,E2 27431.384} C_VEL
LIN {X 0,Y 591.919,Z 792.541,A -85,B 0,C 180,E1 27429.633,E2 27429.633} C_VEL
LIN {X 0,Y 591.916,Z 796.987,A -85,B 0,C 180,E1 27427.873,E2 27427.873} C_VEL
LIN {X 0,Y 591.908,Z 799.837,A -85,B 0,C 180,E1 27426.043,E2 27426.043} C_VEL
LIN {X 0,Y 591.912,Z 800.949,A -85,B 0,C 180,E1 27424.201,E2 27424.201} C_VEL
LIN {X 0,Y 591.912,Z 800.366,A -85,B 0,C 180,E1 27422.431,E2 27422.431} C_VEL
LIN {X 0,Y 591.909,Z 798.139,A -85,B 0,C 180,E1 27420.647,E2 27420.647} C_VEL
LIN {X 0,Y 591.916,Z 794.251,A -85,B 0,C 180,E1 27418.878,E2 27418.878} C_VEL
LIN {X 0,Y 591.93,Z 788.54,A -85,B 0,C 180,E1 27417.087,E2 27417.087} C_VEL
LIN {X 0,Y 591.94,Z 781.131,A -85,B 0,C 180,E1 27415.345,E2 27415.345} C_VEL
LIN {X 0,Y 591.977,Z 772.117,A -85,B 0,C 180,E1 27413.673,E2 27413.673} C_VEL
LIN {X 0,Y 592.024,Z 761.865,A -85,B 0,C 180,E1 27412.124,E2 27412.124} C_VEL
LIN {X 0,Y 592.095,Z 750.195,A -85,B 0,C 180,E1 27410.66,E2 27410.66} C_VEL
LIN {X 0,Y 592.183,Z 737.208,A -85,B 0,C 180,E1 27409.296,E2 27409.296} C_VEL
LIN {X 0,Y 592.286,Z 723.045,A -85,B 0,C 180,E1 27408.05,E2 27408.05} C_VEL
LIN {X 0,Y 592.411,Z 707.045,A -85,B 0,C 180,E1 27406.88,E2 27406.88} C_VEL
LIN {X 0,Y 592.513,Z 689.813,A -85,B 0,C 180,E1 27405.854,E2 27405.854} C_VEL
LIN {X 0,Y 592.648,Z 672.191,A -85,B 0,C 180,E1 27405.019,E2 27405.019} C_VEL
LIN {X 0,Y 592.752,Z 653.919,A -85,B 0,C 180,E1 27404.353,E2 27404.353} C_VEL
LIN {X 0,Y 592.828,Z 635.446,A -85,B 0,C 180,E1 27403.869,E2 27403.869} C_VEL
LIN {X 0,Y 592.884,Z 615.678,A -85,B 0,C 180,E1 27403.543,E2 27403.543} C_VEL
LIN {X 0,Y 592.971,Z 417.982,A -85,B 0,C 180,E1 27401.021,E2 27401.021} C_VEL
LIN {X 0,Y 593.138,Z 361.746,A -85,B 0,C 180,E1 27398.033,E2 27398.033} C_VEL
LIN {X 0,Y 593.485,Z 301.05,A -85,B 0,C 180,E1 27394.703,E2 27394.703} C_VEL
LIN {X 0,Y 593.921,Z 250.032,A -85,B 0,C 180,E1 27391.798,E2 27391.798} C_VEL
LIN {X 0,Y 594.255,Z 231.035,A -85,B 0,C 180,E1 27390.65,E2 27390.65} C_VEL
LIN {X 0,Y 592.008,Z 225.672,A -85,B 0,C 180,E1 27390.106,E2 27390.106} C_VEL
LIN {X 0,Y 592,Z 225.298,A -85,B 0,C 180,E1 27389.549,E2 27389.549} C_VEL
LIN {X 0,Y 591.953,Z 225.308,A -85,B 0,C 180,E1 27386.373,E2 27386.373} C_VEL
LIN {X 0,Y 591.988,Z 225.303,A -85,B 0,C 180,E1 27383.496,E2 27383.496} C_VEL
LIN {X 0,Y 591.96,Z 225.306,A -85,B 0,C 180,E1 27380.361,E2 27380.361} C_VEL
LIN {X 0,Y 591.962,Z 225.306,A -85,B 0,C 180,E1 27377.598,E2 27377.598} C_VEL
LIN {X 0,Y 591.964,Z 225.306,A -85,B 0,C 180,E1 27374.276,E2 27374.276} C_VEL
LIN {X 0,Y 591.964,Z 225.305,A -85,B 0,C 180,E1 27371.397,E2 27371.397} C_VEL
LIN {X 0,Y 591.959,Z 225.305,A -85,B 0,C 180,E1 27368.059,E2 27368.059} C_VEL
LIN {X 0,Y 591.955,Z 225.305,A -85,B 0,C 180,E1 27365.33,E2 27365.33} C_VEL
LIN {X 0,Y 591.969,Z 225.306,A -85,B 0,C 180,E1 27362.032,E2 27362.032} C_VEL
LIN {X 0,Y 591.949,Z 225.305,A -85,B 0,C 180,E1 27359.322,E2 27359.322} C_VEL
LIN {X 0,Y 592.012,Z 225.306,A -85,B 0,C 180,E1 27356.223,E2 27356.223} C_VEL
LIN {X 0,Y 591.946,Z 225.305,A -85,B 0,C 180,E1 27353.296,E2 27353.296} C_VEL
LIN {X 0,Y 592.025,Z 225.305,A -85,B 0,C 180,E1 27350.277,E2 27350.277} C_VEL
LIN {X 0,Y 591.945,Z 225.306,A -85,B 0,C 180,E1 27347.216,E2 27347.216} C_VEL
LIN {X 0,Y 592.012,Z 225.305,A -85,B 0,C 180,E1 27344.222,E2 27344.222} C_VEL
LIN {X 0,Y 591.947,Z 225.306,A -85,B 0,C 180,E1 27341.076,E2 27341.076} C_VEL
LIN {X 0,Y 592.009,Z 225.305,A -85,B 0,C 180,E1 27338.083,E2 27338.083} C_VEL
LIN {X 0,Y 591.951,Z 225.306,A -85,B 0,C 180,E1 27335.022,E2 27335.022} C_VEL
LIN {X 0,Y 591.974,Z 225.306,A -85,B 0,C 180,E1 27332.214,E2 27332.214} C_VEL
LIN {X 0,Y 591.958,Z 225.306,A -85,B 0,C 180,E1 27328.991,E2 27328.991} C_VEL
LIN {X 0,Y 591.962,Z 225.306,A -85,B 0,C 180,E1 27326.2,E2 27326.2} C_VEL
LIN {X 0,Y 591.962,Z 225.306,A -85,B 0,C 180,E1 27322.864,E2 27322.864} C_VEL
LIN {X 0,Y 591.959,Z 225.307,A -85,B 0,C 180,E1 27320.068,E2 27320.068} C_VEL
LIN {X 0,Y 591.963,Z 225.303,A -85,B 0,C 180,E1 27316.705,E2 27316.705} C_VEL
LIN {X 0,Y 591.956,Z 225.3,A -85,B 0,C 180,E1 27313.962,E2 27313.962} C_VEL
LIN {X 0,Y 592.002,Z 225.44,A -85,B 0,C 180,E1 27312.798,E2 27312.798} C_VEL
LIN {X 0,Y 592.399,Z 227.071,A -85,B 0,C 180,E1 27312.593,E2 27312.593} C_VEL
LIN {X 0,Y 594.837,Z 231.545,A -85,B 0,C 180,E1 27312.16,E2 27312.16} C_VEL
LIN {X 0,Y 595.385,Z 233.06,A -85,B 0,C 180,E1 27312.039,E2 27312.039} C_VEL
LIN {X 0,Y 594.937,Z 295.958,A -85,B 0,C 180,E1 27309.096,E2 27309.096} C_VEL
LIN {X 0,Y 594.994,Z 313.169,A -85,B 0,C 180,E1 27308.335,E2 27308.335} C_VEL
LIN {X 0,Y 595.198,Z 324.774,A -85,B 0,C 180,E1 27308.145,E2 27308.145} C_VEL
LIN {X 0,Y 594.706,Z 535.158,A -85,B 0,C 180,E1 27305.08,E2 27305.08} C_VEL
LIN {X 0,Y 594.412,Z 662.55,A -85,B 0,C 180,E1 27303.248,E2 27303.248} C_VEL
LIN {X 0,Y 594.255,Z 686.117,A -85,B 0,C 180,E1 27302.726,E2 27302.726} C_VEL
LIN {X 0,Y 594.111,Z 706.19,A -85,B 0,C 180,E1 27302.123,E2 27302.123} C_VEL
LIN {X 0,Y 593.861,Z 729.437,A -85,B 0,C 180,E1 27301.235,E2 27301.235} C_VEL
LIN {X 0,Y 593.682,Z 749.573,A -85,B 0,C 180,E1 27300.29,E2 27300.29} C_VEL
LIN {X 0,Y 593.398,Z 771.168,A -85,B 0,C 180,E1 27299.084,E2 27299.084} C_VEL
LIN {X 0,Y 593.193,Z 791.465,A -85,B 0,C 180,E1 27297.759,E2 27297.759} C_VEL
LIN {X 0,Y 592.932,Z 811.003,A -85,B 0,C 180,E1 27296.266,E2 27296.266} C_VEL
LIN {X 0,Y 592.683,Z 830.147,A -85,B 0,C 180,E1 27294.592,E2 27294.592} C_VEL
LIN {X 0,Y 592.535,Z 847.278,A -85,B 0,C 180,E1 27292.878,E2 27292.878} C_VEL
LIN {X 0,Y 592.34,Z 863.411,A -85,B 0,C 180,E1 27291.021,E2 27291.021} C_VEL
LIN {X 0,Y 592.184,Z 878.74,A -85,B 0,C 180,E1 27289.001,E2 27289.001} C_VEL
LIN {X 0,Y 592.098,Z 891.386,A -85,B 0,C 180,E1 27287.086,E2 27287.086} C_VEL
LIN {X 0,Y 592.022,Z 902.799,A -85,B 0,C 180,E1 27285.074,E2 27285.074} C_VEL
LIN {X 0,Y 591.982,Z 912.546,A -85,B 0,C 180,E1 27283.08,E2 27283.08} C_VEL
LIN {X 0,Y 591.929,Z 921.341,A -85,B 0,C 180,E1 27280.904,E2 27280.904} C_VEL
LIN {X 0,Y 591.916,Z 928.176,A -85,B 0,C 180,E1 27278.841,E2 27278.841} C_VEL
LIN {X 0,Y 591.914,Z 933.695,A -85,B 0,C 180,E1 27276.664,E2 27276.664} C_VEL
LIN {X 0,Y 591.896,Z 937.437,A -85,B 0,C 180,E1 27274.65,E2 27274.65} C_VEL
LIN {X 0,Y 591.904,Z 939.988,A -85,B 0,C 180,E1 27272.419,E2 27272.419} C_VEL
LIN {X 0,Y 591.897,Z 940.917,A -85,B 0,C 180,E1 27270.386,E2 27270.386} C_VEL
LIN {X 0,Y 591.909,Z 940.322,A -85,B 0,C 180,E1 27268.063,E2 27268.063} C_VEL
LIN {X 0,Y 591.911,Z 938.388,A -85,B 0,C 180,E1 27266.028,E2 27266.028} C_VEL
LIN {X 0,Y 591.915,Z 934.458,A -85,B 0,C 180,E1 27263.695,E2 27263.695} C_VEL
LIN {X 0,Y 591.92,Z 929.802,A -85,B 0,C 180,E1 27261.744,E2 27261.744} C_VEL
LIN {X 0,Y 591.933,Z 922.6,A -85,B 0,C 180,E1 27259.444,E2 27259.444} C_VEL
LIN {X 0,Y 591.964,Z 915.017,A -85,B 0,C 180,E1 27257.493,E2 27257.493} C_VEL
LIN {X 0,Y 592.015,Z 904.872,A -85,B 0,C 180,E1 27255.324,E2 27255.324} C_VEL
LIN {X 0,Y 592.084,Z 894.389,A -85,B 0,C 180,E1 27253.417,E2 27253.417} C_VEL
LIN {X 0,Y 592.188,Z 881.449,A -85,B 0,C 180,E1 27251.39,E2 27251.39} C_VEL
LIN {X 0,Y 592.327,Z 867.209,A -85,B 0,C 180,E1 27249.444,E2 27249.444} C_VEL
LIN {X 0,Y 592.46,Z 851.398,A -85,B 0,C 180,E1 27247.578,E2 27247.578} C_VEL
LIN {X 0,Y 592.666,Z 833.66,A -85,B 0,C 180,E1 27245.744,E2 27245.744} C_VEL
LIN {X 0,Y 592.903,Z 815.532,A -85,B 0,C 180,E1 27244.101,E2 27244.101} C_VEL
LIN {X 0,Y 593.093,Z 796.321,A -85,B 0,C 180,E1 27242.597,E2 27242.597} C_VEL
LIN {X 0,Y 593.377,Z 774.69,A -85,B 0,C 180,E1 27241.133,E2 27241.133} C_VEL
LIN {X 0,Y 593.603,Z 754.637,A -85,B 0,C 180,E1 27239.971,E2 27239.971} C_VEL
LIN {X 0,Y 593.845,Z 732.629,A -85,B 0,C 180,E1 27238.906,E2 27238.906} C_VEL
LIN {X 0,Y 594.051,Z 711.528,A -85,B 0,C 180,E1 27238.058,E2 27238.058} C_VEL
LIN {X 0,Y 594.241,Z 689.321,A -85,B 0,C 180,E1 27237.362,E2 27237.362} C_VEL
LIN {X 0,Y 594.355,Z 668.423,A -85,B 0,C 180,E1 27236.86,E2 27236.86} C_VEL
LIN {X 0,Y 594.491,Z 637.167,A -85,B 0,C 180,E1 27236.368,E2 27236.368} C_VEL
LIN {X 0,Y 594.939,Z 428.104,A -85,B 0,C 180,E1 27233.374,E2 27233.374} C_VEL
LIN {X 0,Y 595.048,Z 313.561,A -85,B 0,C 180,E1 27231.675,E2 27231.675} C_VEL
LIN {X 0,Y 594.862,Z 306.068,A -85,B 0,C 180,E1 27231.365,E2 27231.365} C_VEL
LIN {X 0,Y 595.311,Z 243.84,A -85,B 0,C 180,E1 27228.475,E2 27228.475} C_VEL
LIN {X 0,Y 595.241,Z 232.366,A -85,B 0,C 180,E1 27227.915,E2 27227.915} C_VEL
LIN {X 0,Y 593.858,Z 229.55,A -85,B 0,C 180,E1 27227.657,E2 27227.657} C_VEL
LIN {X 0,Y 592.145,Z 226.234,A -85,B 0,C 180,E1 27227.337,E2 27227.337} C_VEL
LIN {X 0,Y 591.993,Z 225.323,A -85,B 0,C 180,E1 27227.14,E2 27227.14} C_VEL
LIN {X 0,Y 591.952,Z 225.305,A -85,B 0,C 180,E1 27223.965,E2 27223.965} C_VEL
LIN {X 0,Y 591.993,Z 225.305,A -85,B 0,C 180,E1 27220.977,E2 27220.977} C_VEL
LIN {X 0,Y 591.956,Z 225.305,A -85,B 0,C 180,E1 27217.768,E2 27217.768} C_VEL
LIN {X 0,Y 592.004,Z 225.306,A -85,B 0,C 180,E1 27214.81,E2 27214.81} C_VEL
LIN {X 0,Y 591.962,Z 225.303,A -85,B 0,C 180,E1 27211.647,E2 27211.647} C_VEL
LIN {X 0,Y 591.998,Z 225.305,A -85,B 0,C 180,E1 27208.768,E2 27208.768} C_VEL
LIN {X 0,Y 591.972,Z 225.302,A -85,B 0,C 180,E1 27205.585,E2 27205.585} C_VEL
LIN {X 0,Y 592.002,Z 225.305,A -85,B 0,C 180,E1 27202.649,E2 27202.649} C_VEL
LIN {X 0,Y 591.978,Z 225.302,A -85,B 0,C 180,E1 27199.435,E2 27199.435} C_VEL
LIN {X 0,Y 592.024,Z 225.305,A -85,B 0,C 180,E1 27196.382,E2 27196.382} C_VEL
LIN {X 0,Y 591.979,Z 225.301,A -85,B 0,C 180,E1 27193.181,E2 27193.181} C_VEL
LIN {X 0,Y 592.038,Z 225.303,A -85,B 0,C 180,E1 27190.068,E2 27190.068} C_VEL
LIN {X 0,Y 591.981,Z 225.301,A -85,B 0,C 180,E1 27186.985,E2 27186.985} C_VEL
LIN {X 0,Y 592.039,Z 225.302,A -85,B 0,C 180,E1 27183.874,E2 27183.874} C_VEL
LIN {X 0,Y 591.987,Z 225.299,A -85,B 0,C 180,E1 27180.678,E2 27180.678} C_VEL
LIN {X 0,Y 592.039,Z 225.296,A -85,B 0,C 180,E1 27177.484,E2 27177.484} C_VEL
LIN {X 0,Y 592.004,Z 225.302,A -85,B 0,C 180,E1 27174.282,E2 27174.282} C_VEL
LIN {X 0,Y 592.011,Z 225.295,A -85,B 0,C 180,E1 27170.964,E2 27170.964} C_VEL
LIN {X 0,Y 592.008,Z 225.301,A -85,B 0,C 180,E1 27170.164,E2 27170.164} C_VEL
LIN {X 0,Y 591.06,Z 225.426,A -85,B 0,C 180,E1 27169.418,E2 27169.418} C_VEL
LIN {X 0,Y 584.533,Z 226.232,A -85,B 0,C 180,E1 27167.272,E2 27167.272} C_VEL
LIN {X 0,Y 584.07,Z 226.285,A -85,B 0,C 180,E1 27166.781,E2 27166.781} C_VEL
LIN {X 0,Y 584.097,Z 226.292,A -85,B 0,C 180,E1 27163.594,E2 27163.594} C_VEL
LIN {X 0,Y 584.064,Z 226.285,A -85,B 0,C 180,E1 27160.396,E2 27160.396} C_VEL
LIN {X 0,Y 584.09,Z 226.288,A -85,B 0,C 180,E1 27157.241,E2 27157.241} C_VEL
LIN {X 0,Y 584.071,Z 226.289,A -85,B 0,C 180,E1 27154.009,E2 27154.009} C_VEL
LIN {X 0,Y 584.097,Z 226.281,A -85,B 0,C 180,E1 27150.688,E2 27150.688} C_VEL
LIN {X 0,Y 584.094,Z 226.293,A -85,B 0,C 180,E1 27147.37,E2 27147.37} C_VEL
LIN {X 0,Y 584.077,Z 226.286,A -85,B 0,C 180,E1 27144.068,E2 27144.068} C_VEL
LIN {X 0,Y 584.084,Z 226.285,A -85,B 0,C 180,E1 27140.827,E2 27140.827} C_VEL
LIN {X 0,Y 584.08,Z 226.29,A -85,B 0,C 180,E1 27137.691,E2 27137.691} C_VEL
LIN {X 0,Y 584.088,Z 226.285,A -85,B 0,C 180,E1 27134.439,E2 27134.439} C_VEL
LIN {X 0,Y 584.096,Z 226.291,A -85,B 0,C 180,E1 27131.098,E2 27131.098} C_VEL
LIN {X 0,Y 584.087,Z 226.285,A -85,B 0,C 180,E1 27127.796,E2 27127.796} C_VEL
LIN {X 0,Y 584.075,Z 226.288,A -85,B 0,C 180,E1 27124.574,E2 27124.574} C_VEL
LIN {X 0,Y 584.088,Z 226.29,A -85,B 0,C 180,E1 27121.33,E2 27121.33} C_VEL
LIN {X 0,Y 584.078,Z 226.287,A -85,B 0,C 180,E1 27118.084,E2 27118.084} C_VEL
LIN {X 0,Y 584.083,Z 226.292,A -85,B 0,C 180,E1 27114.69,E2 27114.69} C_VEL
LIN {X 0,Y 584.097,Z 226.275,A -85,B 0,C 180,E1 27111.49,E2 27111.49} C_VEL
LIN {X 0,Y 584.065,Z 226.288,A -85,B 0,C 180,E1 27108.258,E2 27108.258} C_VEL
LIN {X 0,Y 584.093,Z 226.287,A -85,B 0,C 180,E1 27105.083,E2 27105.083} C_VEL
LIN {X 0,Y 584.059,Z 226.282,A -85,B 0,C 180,E1 27101.956,E2 27101.956} C_VEL
LIN {X 0,Y 584.094,Z 226.27,A -85,B 0,C 180,E1 27098.764,E2 27098.764} C_VEL
LIN {X 0,Y 584.104,Z 226.541,A -85,B 0,C 180,E1 27098.295,E2 27098.295} C_VEL
LIN {X 0,Y 585.507,Z 229.992,A -85,B 0,C 180,E1 27097.929,E2 27097.929} C_VEL
LIN {X 0,Y 587.404,Z 234.162,A -85,B 0,C 180,E1 27097.532,E2 27097.532} C_VEL
LIN {X 0,Y 586.413,Z 286.938,A -85,B 0,C 180,E1 27094.401,E2 27094.401} C_VEL
LIN {X 0,Y 585.949,Z 343.635,A -85,B 0,C 180,E1 27091.223,E2 27091.223} C_VEL
LIN {X 0,Y 585.495,Z 402.789,A -85,B 0,C 180,E1 27087.995,E2 27087.995} C_VEL
LIN {X 0,Y 585.497,Z 418.177,A -85,B 0,C 180,E1 27087.195,E2 27087.195} C_VEL
LIN {X 0,Y 585.665,Z 448.801,A -85,B 0,C 180,E1 27086.788,E2 27086.788} C_VEL
LIN {X 0,Y 585.338,Z 628.452,A -85,B 0,C 180,E1 27084.45,E2 27084.45} C_VEL
LIN {X 0,Y 585.219,Z 647.407,A -85,B 0,C 180,E1 27084.015,E2 27084.015} C_VEL
LIN {X 0,Y 585.09,Z 665.25,A -85,B 0,C 180,E1 27083.427,E2 27083.427} C_VEL
LIN {X 0,Y 584.906,Z 683.33,A -85,B 0,C 180,E1 27082.635,E2 27082.635} C_VEL
LIN {X 0,Y 584.738,Z 700.305,A -85,B 0,C 180,E1 27081.693,E2 27081.693} C_VEL
LIN {X 0,Y 584.557,Z 716.352,A -85,B 0,C 180,E1 27080.6,E2 27080.6} C_VEL
LIN {X 0,Y 584.387,Z 731.464,A -85,B 0,C 180,E1 27079.353,E2 27079.353} C_VEL
LIN {X 0,Y 584.241,Z 745.586,A -85,B 0,C 180,E1 27077.95,E2 27077.95} C_VEL
LIN {X 0,Y 584.122,Z 758.241,A -85,B 0,C 180,E1 27076.439,E2 27076.439} C_VEL
LIN {X 0,Y 584.039,Z 768.837,A -85,B 0,C 180,E1 27074.914,E2 27074.914} C_VEL
LIN {X 0,Y 583.978,Z 778.156,A -85,B 0,C 180,E1 27073.284,E2 27073.284} C_VEL
LIN {X 0,Y 583.945,Z 786.168,A -85,B 0,C 180,E1 27071.534,E2 27071.534} C_VEL
LIN {X 0,Y 583.921,Z 792.375,A -85,B 0,C 180,E1 27069.765,E2 27069.765} C_VEL
LIN {X 0,Y 583.913,Z 796.883,A -85,B 0,C 180,E1 27067.977,E2 27067.977} C_VEL
LIN {X 0,Y 583.912,Z 799.785,A -85,B 0,C 180,E1 27066.118,E2 27066.118} C_VEL
LIN {X 0,Y 583.912,Z 800.939,A -85,B 0,C 180,E1 27064.247,E2 27064.247} C_VEL
LIN {X 0,Y 583.913,Z 800.403,A -85,B 0,C 180,E1 27062.464,E2 27062.464} C_VEL
LIN {X 0,Y 583.909,Z 798.204,A -85,B 0,C 180,E1 27060.642,E2 27060.642} C_VEL
LIN {X 0,Y 583.918,Z 794.391,A -85,B 0,C 180,E1 27058.862,E2 27058.862} C_VEL
LIN {X 0,Y 583.935,Z 788.692,A -85,B 0,C 180,E1 27057.035,E2 27057.035} C_VEL
LIN {X 0,Y 583.957,Z 781.336,A -85,B 0,C 180,E1 27055.27,E2 27055.27} C_VEL
LIN {X 0,Y 584.014,Z 772.38,A -85,B 0,C 180,E1 27053.576,E2 27053.576} C_VEL
LIN {X 0,Y 584.093,Z 761.756,A -85,B 0,C 180,E1 27051.945,E2 27051.945} C_VEL
LIN {X 0,Y 584.198,Z 750.027,A -85,B 0,C 180,E1 27050.457,E2 27050.457} C_VEL
LIN {X 0,Y 584.339,Z 736.815,A -85,B 0,C 180,E1 27049.056,E2 27049.056} C_VEL
LIN {X 0,Y 584.5,Z 722.162,A -85,B 0,C 180,E1 27047.759,E2 27047.759} C_VEL
LIN {X 0,Y 584.683,Z 705.92,A -85,B 0,C 180,E1 27046.573,E2 27046.573} C_VEL
LIN {X 0,Y 584.842,Z 689.166,A -85,B 0,C 180,E1 27045.575,E2 27045.575} C_VEL
LIN {X 0,Y 585.033,Z 672.083,A -85,B 0,C 180,E1 27044.759,E2 27044.759} C_VEL
LIN {X 0,Y 585.189,Z 653.901,A -85,B 0,C 180,E1 27044.089,E2 27044.089} C_VEL
LIN {X 0,Y 585.305,Z 635.294,A -85,B 0,C 180,E1 27043.596,E2 27043.596} C_VEL
LIN {X 0,Y 585.388,Z 615.42,A -85,B 0,C 180,E1 27043.267,E2 27043.267} C_VEL
LIN {X 0,Y 585.6,Z 418.931,A -85,B 0,C 180,E1 27040.729,E2 27040.729} C_VEL
LIN {X 0,Y 585.416,Z 416.628,A -85,B 0,C 180,E1 27040.66,E2 27040.66} C_VEL
LIN {X 0,Y 585.8,Z 359.159,A -85,B 0,C 180,E1 27037.541,E2 27037.541} C_VEL
LIN {X 0,Y 586.319,Z 299.927,A -85,B 0,C 180,E1 27034.246,E2 27034.246} C_VEL
LIN {X 0,Y 587.182,Z 254.65,A -85,B 0,C 180,E1 27031.574,E2 27031.574} C_VEL
LIN {X 0,Y 587.625,Z 234.564,A -85,B 0,C 180,E1 27030.354,E2 27030.354} C_VEL
LIN {X 0,Y 584.182,Z 227.017,A -85,B 0,C 180,E1 27029.589,E2 27029.589} C_VEL
LIN {X 0,Y 584.086,Z 226.301,A -85,B 0,C 180,E1 27029.39,E2 27029.39} C_VEL
LIN {X 0,Y 584.013,Z 226.297,A -85,B 0,C 180,E1 27026.212,E2 27026.212} C_VEL
LIN {X 0,Y 584.093,Z 226.292,A -85,B 0,C 180,E1 27023.185,E2 27023.185} C_VEL
LIN {X 0,Y 584.012,Z 226.295,A -85,B 0,C 180,E1 27020.128,E2 27020.128} C_VEL
LIN {X 0,Y 584.075,Z 226.295,A -85,B 0,C 180,E1 27017.123,E2 27017.123} C_VEL
LIN {X 0,Y 584.014,Z 226.295,A -85,B 0,C 180,E1 27014.07,E2 27014.07} C_VEL
LIN {X 0,Y 584.049,Z 226.295,A -85,B 0,C 180,E1 27011.154,E2 27011.154} C_VEL
LIN {X 0,Y 584.016,Z 226.293,A -85,B 0,C 180,E1 27007.971,E2 27007.971} C_VEL
LIN {X 0,Y 584.025,Z 226.294,A -85,B 0,C 180,E1 27005.206,E2 27005.206} C_VEL
LIN {X 0,Y 584.018,Z 226.295,A -85,B 0,C 180,E1 27001.864,E2 27001.864} C_VEL
LIN {X 0,Y 584.02,Z 226.293,A -85,B 0,C 180,E1 26999.117,E2 26999.117} C_VEL
LIN {X 0,Y 584.024,Z 226.295,A -85,B 0,C 180,E1 26995.778,E2 26995.778} C_VEL
LIN {X 0,Y 584.021,Z 226.294,A -85,B 0,C 180,E1 26992.919,E2 26992.919} C_VEL
LIN {X 0,Y 584.017,Z 226.295,A -85,B 0,C 180,E1 26989.544,E2 26989.544} C_VEL
LIN {X 0,Y 584.029,Z 226.295,A -85,B 0,C 180,E1 26986.637,E2 26986.637} C_VEL
LIN {X 0,Y 584.019,Z 226.295,A -85,B 0,C 180,E1 26983.387,E2 26983.387} C_VEL
LIN {X 0,Y 584.02,Z 226.295,A -85,B 0,C 180,E1 26980.601,E2 26980.601} C_VEL
LIN {X 0,Y 584.02,Z 226.294,A -85,B 0,C 180,E1 26977.237,E2 26977.237} C_VEL
LIN {X 0,Y 584.02,Z 226.295,A -85,B 0,C 180,E1 26974.441,E2 26974.441} C_VEL
LIN {X 0,Y 584.026,Z 226.295,A -85,B 0,C 180,E1 26971.132,E2 26971.132} C_VEL
LIN {X 0,Y 584.021,Z 226.295,A -85,B 0,C 180,E1 26968.292,E2 26968.292} C_VEL
LIN {X 0,Y 584.021,Z 226.296,A -85,B 0,C 180,E1 26964.883,E2 26964.883} C_VEL
LIN {X 0,Y 584.035,Z 226.296,A -85,B 0,C 180,E1 26961.951,E2 26961.951} C_VEL
LIN {X 0,Y 584.022,Z 226.297,A -85,B 0,C 180,E1 26958.725,E2 26958.725} C_VEL
LIN {X 0,Y 584.031,Z 226.293,A -85,B 0,C 180,E1 26955.831,E2 26955.831} C_VEL
LIN {X 0,Y 584.091,Z 226.471,A -85,B 0,C 180,E1 26953.464,E2 26953.464} C_VEL
LIN {X 0,Y 584.399,Z 227.695,A -85,B 0,C 180,E1 26953.289,E2 26953.289} C_VEL
LIN {X 0,Y 589.152,Z 236.503,A -85,B 0,C 180,E1 26952.418,E2 26952.418} C_VEL
LIN {X 0,Y 588.491,Z 298.494,A -85,B 0,C 180,E1 26949.488,E2 26949.488} C_VEL
LIN {X 0,Y 588.519,Z 313.215,A -85,B 0,C 180,E1 26948.834,E2 26948.834} C_VEL
LIN {X 0,Y 588.923,Z 318.839,A -85,B 0,C 180,E1 26948.716,E2 26948.716} C_VEL
LIN {X 0,Y 588.173,Z 530.528,A -85,B 0,C 180,E1 26945.596,E2 26945.596} C_VEL
LIN {X 0,Y 587.709,Z 662.657,A -85,B 0,C 180,E1 26943.675,E2 26943.675} C_VEL
LIN {X 0,Y 587.468,Z 686.337,A -85,B 0,C 180,E1 26943.146,E2 26943.146} C_VEL
LIN {X 0,Y 587.25,Z 706.947,A -85,B 0,C 180,E1 26942.519,E2 26942.519} C_VEL
LIN {X 0,Y 586.875,Z 730.152,A -85,B 0,C 180,E1 26941.617,E2 26941.617} C_VEL
LIN {X 0,Y 586.588,Z 751.569,A -85,B 0,C 180,E1 26940.595,E2 26940.595} C_VEL
LIN {X 0,Y 586.172,Z 772.061,A -85,B 0,C 180,E1 26939.421,E2 26939.421} C_VEL
LIN {X 0,Y 585.845,Z 792.35,A -85,B 0,C 180,E1 26938.072,E2 26938.072} C_VEL
LIN {X 0,Y 585.468,Z 810.939,A -85,B 0,C 180,E1 26936.633,E2 26936.633} C_VEL
LIN {X 0,Y 585.122,Z 830.125,A -85,B 0,C 180,E1 26934.934,E2 26934.934} C_VEL
LIN {X 0,Y 584.858,Z 847.172,A -85,B 0,C 180,E1 26933.207,E2 26933.207} C_VEL
LIN {X 0,Y 584.572,Z 863.001,A -85,B 0,C 180,E1 26931.364,E2 26931.364} C_VEL
LIN {X 0,Y 584.367,Z 877.922,A -85,B 0,C 180,E1 26929.385,E2 26929.385} C_VEL
LIN {X 0,Y 584.221,Z 890.745,A -85,B 0,C 180,E1 26927.426,E2 26927.426} C_VEL
LIN {X 0,Y 584.093,Z 902.8,A -85,B 0,C 180,E1 26925.284,E2 26925.284} C_VEL
LIN {X 0,Y 584.023,Z 912.546,A -85,B 0,C 180,E1 26923.261,E2 26923.261} C_VEL
LIN {X 0,Y 583.949,Z 921.342,A -85,B 0,C 180,E1 26921.055,E2 26921.055} C_VEL
LIN {X 0,Y 583.941,Z 927.872,A -85,B 0,C 180,E1 26919.062,E2 26919.062} C_VEL
LIN {X 0,Y 583.915,Z 933.636,A -85,B 0,C 180,E1 26916.784,E2 26916.784} C_VEL
LIN {X 0,Y 583.899,Z 937.437,A -85,B 0,C 180,E1 26914.714,E2 26914.714} C_VEL
LIN {X 0,Y 583.907,Z 939.988,A -85,B 0,C 180,E1 26912.452,E2 26912.452} C_VEL
LIN {X 0,Y 583.897,Z 940.917,A -85,B 0,C 180,E1 26910.391,E2 26910.391} C_VEL
LIN {X 0,Y 583.91,Z 940.323,A -85,B 0,C 180,E1 26908.036,E2 26908.036} C_VEL
LIN {X 0,Y 583.911,Z 938.389,A -85,B 0,C 180,E1 26905.973,E2 26905.973} C_VEL
LIN {X 0,Y 583.92,Z 934.458,A -85,B 0,C 180,E1 26903.609,E2 26903.609} C_VEL
LIN {X 0,Y 583.924,Z 929.802,A -85,B 0,C 180,E1 26901.63,E2 26901.63} C_VEL
LIN {X 0,Y 583.946,Z 922.759,A -85,B 0,C 180,E1 26899.342,E2 26899.342} C_VEL
LIN {X 0,Y 583.995,Z 915.102,A -85,B 0,C 180,E1 26897.34,E2 26897.34} C_VEL
LIN {X 0,Y 584.068,Z 904.874,A -85,B 0,C 180,E1 26895.12,E2 26895.12} C_VEL
LIN {X 0,Y 584.175,Z 894.39,A -85,B 0,C 180,E1 26893.186,E2 26893.186} C_VEL
LIN {X 0,Y 584.329,Z 881.442,A -85,B 0,C 180,E1 26891.129,E2 26891.129} C_VEL
LIN {X 0,Y 584.547,Z 867.21,A -85,B 0,C 180,E1 26889.158,E2 26889.158} C_VEL
LIN {X 0,Y 584.761,Z 851.399,A -85,B 0,C 180,E1 26887.267,E2 26887.267} C_VEL
LIN {X 0,Y 585.061,Z 833.489,A -85,B 0,C 180,E1 26885.392,E2 26885.392} C_VEL
LIN {X 0,Y 585.431,Z 815.24,A -85,B 0,C 180,E1 26883.721,E2 26883.721} C_VEL
LIN {X 0,Y 585.729,Z 796.323,A -85,B 0,C 180,E1 26882.223,E2 26882.223} C_VEL
LIN {X 0,Y 586.143,Z 774.693,A -85,B 0,C 180,E1 26880.743,E2 26880.743} C_VEL
LIN {X 0,Y 586.504,Z 754.825,A -85,B 0,C 180,E1 26879.58,E2 26879.58} C_VEL
LIN {X 0,Y 586.849,Z 733.205,A -85,B 0,C 180,E1 26878.519,E2 26878.519} C_VEL
LIN {X 0,Y 587.152,Z 712.499,A -85,B 0,C 180,E1 26877.675,E2 26877.675} C_VEL
LIN {X 0,Y 587.448,Z 689.842,A -85,B 0,C 180,E1 26876.951,E2 26876.951} C_VEL
LIN {X 0,Y 587.623,Z 668.931,A -85,B 0,C 180,E1 26876.442,E2 26876.442} C_VEL
LIN {X 0,Y 587.824,Z 638.052,A -85,B 0,C 180,E1 26875.947,E2 26875.947} C_VEL
LIN {X 0,Y 588.511,Z 428.953,A -85,B 0,C 180,E1 26872.92,E2 26872.92} C_VEL
LIN {X 0,Y 588.754,Z 314.932,A -85,B 0,C 180,E1 26871.211,E2 26871.211} C_VEL
LIN {X 0,Y 588.372,Z 309.947,A -85,B 0,C 180,E1 26871.04,E2 26871.04} C_VEL
LIN {X 0,Y 589.046,Z 247.08,A -85,B 0,C 180,E1 26868.091,E2 26868.091} C_VEL
LIN {X 0,Y 589.152,Z 236.503,A -85,B 0,C 180,E1 26867.582,E2 26867.582} C_VEL
LIN {X 0,Y 585.635,Z 230.1,A -85,B 0,C 180,E1 26866.947,E2 26866.947} C_VEL
LIN {X 0,Y 584.12,Z 226.631,A -85,B 0,C 180,E1 26866.582,E2 26866.582} C_VEL
LIN {X 0,Y 584.017,Z 226.273,A -85,B 0,C 180,E1 26866.101,E2 26866.101} C_VEL
LIN {X 0,Y 584.022,Z 226.285,A -85,B 0,C 180,E1 26863.313,E2 26863.313} C_VEL
LIN {X 0,Y 584.03,Z 226.293,A -85,B 0,C 180,E1 26860.069,E2 26860.069} C_VEL
LIN {X 0,Y 584.029,Z 226.295,A -85,B 0,C 180,E1 26857.181,E2 26857.181} C_VEL
LIN {X 0,Y 584.027,Z 226.294,A -85,B 0,C 180,E1 26853.807,E2 26853.807} C_VEL
LIN {X 0,Y 584.047,Z 226.293,A -85,B 0,C 180,E1 26850.903,E2 26850.903} C_VEL
LIN {X 0,Y 584.032,Z 226.293,A -85,B 0,C 180,E1 26847.642,E2 26847.642} C_VEL
LIN {X 0,Y 584.069,Z 226.292,A -85,B 0,C 180,E1 26844.63,E2 26844.63} C_VEL
LIN {X 0,Y 584.037,Z 226.291,A -85,B 0,C 180,E1 26841.492,E2 26841.492} C_VEL
LIN {X 0,Y 584.077,Z 226.293,A -85,B 0,C 180,E1 26838.463,E2 26838.463} C_VEL
LIN {X 0,Y 584.041,Z 226.29,A -85,B 0,C 180,E1 26835.287,E2 26835.287} C_VEL
LIN {X 0,Y 584.095,Z 226.294,A -85,B 0,C 180,E1 26832.155,E2 26832.155} C_VEL
LIN {X 0,Y 584.042,Z 226.29,A -85,B 0,C 180,E1 26828.956,E2 26828.956} C_VEL
LIN {X 0,Y 584.101,Z 226.287,A -85,B 0,C 180,E1 26825.797,E2 26825.797} C_VEL
LIN {X 0,Y 584.05,Z 226.291,A -85,B 0,C 180,E1 26822.65,E2 26822.65} C_VEL
LIN {X 0,Y 584.092,Z 226.286,A -85,B 0,C 180,E1 26819.412,E2 26819.412} C_VEL
LIN {X 0,Y 584.074,Z 226.291,A -85,B 0,C 180,E1 26816.172,E2 26816.172} C_VEL
LIN {X 0,Y 584.065,Z 226.287,A -85,B 0,C 180,E1 26812.92,E2 26812.92} C_VEL
LIN {X 0,Y 584.098,Z 226.293,A -85,B 0,C 180,E1 26809.746,E2 26809.746} C_VEL
LIN {X 0,Y 584.07,Z 226.285,A -85,B 0,C 180,E1 26806.781,E2 26806.781} C_VEL
LIN {X 0,Y 583.054,Z 226.419,A -85,B 0,C 180,E1 26806.026,E2 26806.026} C_VEL
LIN {X 0,Y 576.673,Z 227.218,A -85,B 0,C 180,E1 26803.905,E2 26803.905} C_VEL
LIN {X 0,Y 576.154,Z 227.278,A -85,B 0,C 180,E1 26803.353,E2 26803.353} C_VEL
LIN {X 0,Y 576.129,Z 227.275,A -85,B 0,C 180,E1 26800.114,E2 26800.114} C_VEL
LIN {X 0,Y 576.158,Z 227.272,A -85,B 0,C 180,E1 26796.801,E2 26796.801} C_VEL
LIN {X 0,Y 576.157,Z 227.283,A -85,B 0,C 180,E1 26793.514,E2 26793.514} C_VEL
LIN {X 0,Y 576.134,Z 227.272,A -85,B 0,C 180,E1 26790.197,E2 26790.197} C_VEL
LIN {X 0,Y 576.149,Z 227.275,A -85,B 0,C 180,E1 26786.952,E2 26786.952} C_VEL
LIN {X 0,Y 576.141,Z 227.278,A -85,B 0,C 180,E1 26783.717,E2 26783.717} C_VEL
LIN {X 0,Y 576.155,Z 227.269,A -85,B 0,C 180,E1 26780.401,E2 26780.401} C_VEL
LIN {X 0,Y 576.151,Z 227.278,A -85,B 0,C 180,E1 26777.084,E2 26777.084} C_VEL
LIN {X 0,Y 576.143,Z 227.277,A -85,B 0,C 180,E1 26773.786,E2 26773.786} C_VEL
LIN {X 0,Y 576.141,Z 227.276,A -85,B 0,C 180,E1 26770.526,E2 26770.526} C_VEL
LIN {X 0,Y 576.155,Z 227.279,A -85,B 0,C 180,E1 26767.2,E2 26767.2} C_VEL
LIN {X 0,Y 576.158,Z 227.272,A -85,B 0,C 180,E1 26763.853,E2 26763.853} C_VEL
LIN {X 0,Y 576.135,Z 227.277,A -85,B 0,C 180,E1 26760.564,E2 26760.564} C_VEL
LIN {X 0,Y 576.151,Z 227.279,A -85,B 0,C 180,E1 26757.313,E2 26757.313} C_VEL
LIN {X 0,Y 576.133,Z 227.276,A -85,B 0,C 180,E1 26754.07,E2 26754.07} C_VEL
LIN {X 0,Y 576.148,Z 227.274,A -85,B 0,C 180,E1 26750.711,E2 26750.711} C_VEL
LIN {X 0,Y 576.157,Z 227.273,A -85,B 0,C 180,E1 26747.368,E2 26747.368} C_VEL
LIN {X 0,Y 576.123,Z 227.281,A -85,B 0,C 180,E1 26744.165,E2 26744.165} C_VEL
LIN {X 0,Y 576.156,Z 227.275,A -85,B 0,C 180,E1 26740.905,E2 26740.905} C_VEL
LIN {X 0,Y 576.181,Z 227.453,A -85,B 0,C 180,E1 26738.86,E2 26738.86} C_VEL
LIN {X 0,Y 577.044,Z 230.06,A -85,B 0,C 180,E1 26738.571,E2 26738.571} C_VEL
LIN {X 0,Y 580.644,Z 238.063,A -85,B 0,C 180,E1 26737.795,E2 26737.795} C_VEL
LIN {X 0,Y 579.447,Z 291.298,A -85,B 0,C 180,E1 26734.603,E2 26734.603} C_VEL
LIN {X 0,Y 578.707,Z 340.283,A -85,B 0,C 180,E1 26731.783,E2 26731.783} C_VEL
LIN {X 0,Y 578.106,Z 398.398,A -85,B 0,C 180,E1 26728.564,E2 26728.564} C_VEL
LIN {X 0,Y 578.02,Z 418.064,A -85,B 0,C 180,E1 26727.516,E2 26727.516} C_VEL
LIN {X 0,Y 578.362,Z 425.978,A -85,B 0,C 180,E1 26727.395,E2 26727.395} C_VEL
LIN {X 0,Y 577.841,Z 628.386,A -85,B 0,C 180,E1 26724.73,E2 26724.73} C_VEL
LIN {X 0,Y 577.686,Z 647.377,A -85,B 0,C 180,E1 26724.29,E2 26724.29} C_VEL
LIN {X 0,Y 577.506,Z 665.334,A -85,B 0,C 180,E1 26723.689,E2 26723.689} C_VEL
LIN {X 0,Y 577.264,Z 683.414,A -85,B 0,C 180,E1 26722.887,E2 26722.887} C_VEL
LIN {X 0,Y 577.034,Z 700.387,A -85,B 0,C 180,E1 26721.933,E2 26721.933} C_VEL
LIN {X 0,Y 576.791,Z 716.429,A -85,B 0,C 180,E1 26720.824,E2 26720.824} C_VEL
LIN {X 0,Y 576.562,Z 731.534,A -85,B 0,C 180,E1 26719.56,E2 26719.56} C_VEL
LIN {X 0,Y 576.368,Z 745.187,A -85,B 0,C 180,E1 26718.189,E2 26718.189} C_VEL
LIN {X 0,Y 576.204,Z 757.903,A -85,B 0,C 180,E1 26716.658,E2 26716.658} C_VEL
LIN {X 0,Y 576.084,Z 769.173,A -85,B 0,C 180,E1 26715.014,E2 26715.014} C_VEL
LIN {X 0,Y 576.001,Z 778.45,A -85,B 0,C 180,E1 26713.358,E2 26713.358} C_VEL
LIN {X 0,Y 575.955,Z 786.396,A -85,B 0,C 180,E1 26711.583,E2 26711.583} C_VEL
LIN {X 0,Y 575.925,Z 792.545,A -85,B 0,C 180,E1 26709.79,E2 26709.79} C_VEL
LIN {X 0,Y 575.914,Z 796.999,A -85,B 0,C 180,E1 26707.977,E2 26707.977} C_VEL
LIN {X 0,Y 575.913,Z 799.794,A -85,B 0,C 180,E1 26706.141,E2 26706.141} C_VEL
LIN {X 0,Y 575.912,Z 800.933,A -85,B 0,C 180,E1 26704.278,E2 26704.278} C_VEL
LIN {X 0,Y 575.913,Z 800.364,A -85,B 0,C 180,E1 26702.385,E2 26702.385} C_VEL
LIN {X 0,Y 575.909,Z 798.169,A -85,B 0,C 180,E1 26700.574,E2 26700.574} C_VEL
LIN {X 0,Y 575.922,Z 794.237,A -85,B 0,C 180,E1 26698.73,E2 26698.73} C_VEL
LIN {X 0,Y 575.94,Z 788.801,A -85,B 0,C 180,E1 26696.969,E2 26696.969} C_VEL
LIN {X 0,Y 575.977,Z 781.448,A -85,B 0,C 180,E1 26695.173,E2 26695.173} C_VEL
LIN {X 0,Y 576.052,Z 772.57,A -85,B 0,C 180,E1 26693.464,E2 26693.464} C_VEL
LIN {X 0,Y 576.158,Z 762.082,A -85,B 0,C 180,E1 26691.824,E2 26691.824} C_VEL
LIN {X 0,Y 576.298,Z 750.488,A -85,B 0,C 180,E1 26690.324,E2 26690.324} C_VEL
LIN {X 0,Y 576.483,Z 737.371,A -85,B 0,C 180,E1 26688.905,E2 26688.905} C_VEL
LIN {X 0,Y 576.698,Z 722.841,A -85,B 0,C 180,E1 26687.592,E2 26687.592} C_VEL
LIN {X 0,Y 576.946,Z 706.816,A -85,B 0,C 180,E1 26686.392,E2 26686.392} C_VEL
LIN {X 0,Y 577.173,Z 689.912,A -85,B 0,C 180,E1 26685.361,E2 26685.361} C_VEL
LIN {X 0,Y 577.428,Z 671.935,A -85,B 0,C 180,E1 26684.489,E2 26684.489} C_VEL
LIN {X 0,Y 577.638,Z 653.624,A -85,B 0,C 180,E1 26683.809,E2 26683.809} C_VEL
LIN {X 0,Y 577.796,Z 635.089,A -85,B 0,C 180,E1 26683.315,E2 26683.315} C_VEL
LIN {X 0,Y 577.903,Z 615.027,A -85,B 0,C 180,E1 26682.981,E2 26682.981} C_VEL
LIN {X 0,Y 578.236,Z 419.799,A -85,B 0,C 180,E1 26680.427,E2 26680.427} C_VEL
LIN {X 0,Y 577.945,Z 416.191,A -85,B 0,C 180,E1 26680.317,E2 26680.317} C_VEL
LIN {X 0,Y 578.486,Z 358.403,A -85,B 0,C 180,E1 26677.138,E2 26677.138} C_VEL
LIN {X 0,Y 579.213,Z 306.41,A -85,B 0,C 180,E1 26674.186,E2 26674.186} C_VEL
LIN {X 0,Y 580.64,Z 251.489,A -85,B 0,C 180,E1 26670.873,E2 26670.873} C_VEL
LIN {X 0,Y 580.921,Z 238.288,A -85,B 0,C 180,E1 26670.056,E2 26670.056} C_VEL
LIN {X 0,Y 576.188,Z 227.741,A -85,B 0,C 180,E1 26668.956,E2 26668.956} C_VEL
LIN {X 0,Y 576.095,Z 227.286,A -85,B 0,C 180,E1 26668.734,E2 26668.734} C_VEL
LIN {X 0,Y 576.087,Z 227.287,A -85,B 0,C 180,E1 26665.825,E2 26665.825} C_VEL
LIN {X 0,Y 576.084,Z 227.284,A -85,B 0,C 180,E1 26662.447,E2 26662.447} C_VEL
LIN {X 0,Y 576.092,Z 227.284,A -85,B 0,C 180,E1 26659.57,E2 26659.57} C_VEL
LIN {X 0,Y 576.08,Z 227.285,A -85,B 0,C 180,E1 26656.226,E2 26656.226} C_VEL
LIN {X 0,Y 576.088,Z 227.284,A -85,B 0,C 180,E1 26653.448,E2 26653.448} C_VEL
LIN {X 0,Y 576.081,Z 227.283,A -85,B 0,C 180,E1 26650.096,E2 26650.096} C_VEL
LIN {X 0,Y 576.094,Z 227.282,A -85,B 0,C 180,E1 26647.178,E2 26647.178} C_VEL
LIN {X 0,Y 576.078,Z 227.284,A -85,B 0,C 180,E1 26643.881,E2 26643.881} C_VEL
LIN {X 0,Y 576.094,Z 227.284,A -85,B 0,C 180,E1 26640.994,E2 26640.994} C_VEL
LIN {X 0,Y 576.077,Z 227.284,A -85,B 0,C 180,E1 26637.712,E2 26637.712} C_VEL
LIN {X 0,Y 576.094,Z 227.284,A -85,B 0,C 180,E1 26634.822,E2 26634.822} C_VEL
LIN {X 0,Y 576.075,Z 227.283,A -85,B 0,C 180,E1 26631.516,E2 26631.516} C_VEL
LIN {X 0,Y 576.101,Z 227.284,A -85,B 0,C 180,E1 26628.588,E2 26628.588} C_VEL
LIN {X 0,Y 576.072,Z 227.282,A -85,B 0,C 180,E1 26625.321,E2 26625.321} C_VEL
LIN {X 0,Y 576.101,Z 227.284,A -85,B 0,C 180,E1 26622.423,E2 26622.423} C_VEL
LIN {X 0,Y 576.074,Z 227.283,A -85,B 0,C 180,E1 26619.157,E2 26619.157} C_VEL
LIN {X 0,Y 576.091,Z 227.283,A -85,B 0,C 180,E1 26616.364,E2 26616.364} C_VEL
LIN {X 0,Y 576.079,Z 227.285,A -85,B 0,C 180,E1 26613.064,E2 26613.064} C_VEL
LIN {X 0,Y 576.1,Z 227.285,A -85,B 0,C 180,E1 26610.125,E2 26610.125} C_VEL
LIN {X 0,Y 576.078,Z 227.285,A -85,B 0,C 180,E1 26606.857,E2 26606.857} C_VEL
LIN {X 0,Y 576.114,Z 227.286,A -85,B 0,C 180,E1 26603.837,E2 26603.837} C_VEL
LIN {X 0,Y 576.078,Z 227.285,A -85,B 0,C 180,E1 26600.691,E2 26600.691} C_VEL
LIN {X 0,Y 576.1,Z 227.287,A -85,B 0,C 180,E1 26597.804,E2 26597.804} C_VEL
LIN {X 0,Y 576.077,Z 227.274,A -85,B 0,C 180,E1 26594.521,E2 26594.521} C_VEL
LIN {X 0,Y 576.132,Z 227.664,A -85,B 0,C 180,E1 26594.116,E2 26594.116} C_VEL
LIN {X 0,Y 577.458,Z 230.833,A -85,B 0,C 180,E1 26593.778,E2 26593.778} C_VEL
LIN {X 0,Y 578.671,Z 232.422,A -85,B 0,C 180,E1 26593.582,E2 26593.582} C_VEL
LIN {X 0,Y 582.952,Z 240.646,A -85,B 0,C 180,E1 26592.77,E2 26592.77} C_VEL
LIN {X 0,Y 582.056,Z 302.125,A -85,B 0,C 180,E1 26589.838,E2 26589.838} C_VEL
LIN {X 0,Y 582.099,Z 313.333,A -85,B 0,C 180,E1 26589.343,E2 26589.343} C_VEL
LIN {X 0,Y 582.671,Z 319.699,A -85,B 0,C 180,E1 26589.197,E2 26589.197} C_VEL
LIN {X 0,Y 581.66,Z 531.292,A -85,B 0,C 180,E1 26586.046,E2 26586.046} C_VEL
LIN {X 0,Y 581.04,Z 662.765,A -85,B 0,C 180,E1 26584.113,E2 26584.113} C_VEL
LIN {X 0,Y 580.715,Z 686.532,A -85,B 0,C 180,E1 26583.577,E2 26583.577} C_VEL
LIN {X 0,Y 580.418,Z 707.758,A -85,B 0,C 180,E1 26582.922,E2 26582.922} C_VEL
LIN {X 0,Y 579.953,Z 729.444,A -85,B 0,C 180,E1 26582.072,E2 26582.072} C_VEL
LIN {X 0,Y 579.554,Z 749.579,A -85,B 0,C 180,E1 26581.11,E2 26581.11} C_VEL
LIN {X 0,Y 579.022,Z 771.173,A -85,B 0,C 180,E1 26579.878,E2 26579.878} C_VEL
LIN {X 0,Y 578.577,Z 791.211,A -85,B 0,C 180,E1 26578.542,E2 26578.542} C_VEL
LIN {X 0,Y 578.04,Z 810.684,A -85,B 0,C 180,E1 26577.024,E2 26577.024} C_VEL
LIN {X 0,Y 577.576,Z 830.366,A -85,B 0,C 180,E1 26575.258,E2 26575.258} C_VEL
LIN {X 0,Y 577.19,Z 847.687,A -85,B 0,C 180,E1 26573.478,E2 26573.478} C_VEL
LIN {X 0,Y 576.81,Z 863.854,A -85,B 0,C 180,E1 26571.559,E2 26571.559} C_VEL
LIN {X 0,Y 576.512,Z 879.341,A -85,B 0,C 180,E1 26569.449,E2 26569.449} C_VEL
LIN {X 0,Y 576.317,Z 892.363,A -85,B 0,C 180,E1 26567.408,E2 26567.408} C_VEL
LIN {X 0,Y 576.151,Z 903.843,A -85,B 0,C 180,E1 26565.293,E2 26565.293} C_VEL
LIN {X 0,Y 576.051,Z 913.884,A -85,B 0,C 180,E1 26563.142,E2 26563.142} C_VEL
LIN {X 0,Y 575.963,Z 922.055,A -85,B 0,C 180,E1 26561.007,E2 26561.007} C_VEL
LIN {X 0,Y 575.928,Z 929.043,A -85,B 0,C 180,E1 26558.787,E2 26558.787} C_VEL
LIN {X 0,Y 575.918,Z 934.049,A -85,B 0,C 180,E1 26556.679,E2 26556.679} C_VEL
LIN {X 0,Y 575.9,Z 937.914,A -85,B 0,C 180,E1 26554.48,E2 26554.48} C_VEL
LIN {X 0,Y 575.904,Z 940.123,A -85,B 0,C 180,E1 26552.287,E2 26552.287} C_VEL
LIN {X 0,Y 575.91,Z 940.984,A -85,B 0,C 180,E1 26550.098,E2 26550.098} C_VEL
LIN {X 0,Y 575.908,Z 940.188,A -85,B 0,C 180,E1 26547.81,E2 26547.81} C_VEL
LIN {X 0,Y 575.904,Z 938.048,A -85,B 0,C 180,E1 26545.618,E2 26545.618} C_VEL
LIN {X 0,Y 575.923,Z 934.252,A -85,B 0,C 180,E1 26543.42,E2 26543.42} C_VEL
LIN {X 0,Y 575.925,Z 929.293,A -85,B 0,C 180,E1 26541.312,E2 26541.312} C_VEL
LIN {X 0,Y 575.96,Z 922.404,A -85,B 0,C 180,E1 26539.092,E2 26539.092} C_VEL
LIN {X 0,Y 576.041,Z 914.694,A -85,B 0,C 180,E1 26537.06,E2 26537.06} C_VEL
LIN {X 0,Y 576.142,Z 904.354,A -85,B 0,C 180,E1 26534.807,E2 26534.807} C_VEL
LIN {X 0,Y 576.297,Z 893.231,A -85,B 0,C 180,E1 26532.741,E2 26532.741} C_VEL
LIN {X 0,Y 576.48,Z 880.744,A -85,B 0,C 180,E1 26530.758,E2 26530.758} C_VEL
LIN {X 0,Y 576.78,Z 866.379,A -85,B 0,C 180,E1 26528.757,E2 26528.757} C_VEL
LIN {X 0,Y 577.092,Z 851.214,A -85,B 0,C 180,E1 26526.926,E2 26526.926} C_VEL
LIN {X 0,Y 577.487,Z 833.108,A -85,B 0,C 180,E1 26525.009,E2 26525.009} C_VEL
LIN {X 0,Y 577.977,Z 814.883,A -85,B 0,C 180,E1 26523.325,E2 26523.325} C_VEL
LIN {X 0,Y 578.43,Z 795.671,A -85,B 0,C 180,E1 26521.791,E2 26521.791} C_VEL
LIN {X 0,Y 578.947,Z 774.137,A -85,B 0,C 180,E1 26520.307,E2 26520.307} C_VEL
LIN {X 0,Y 579.471,Z 753.816,A -85,B 0,C 180,E1 26519.114,E2 26519.114} C_VEL
LIN {X 0,Y 579.905,Z 731.651,A -85,B 0,C 180,E1 26518.026,E2 26518.026} C_VEL
LIN {X 0,Y 580.403,Z 709.227,A -85,B 0,C 180,E1 26517.127,E2 26517.127} C_VEL
LIN {X 0,Y 580.707,Z 687.381,A -85,B 0,C 180,E1 26516.447,E2 26516.447} C_VEL
LIN {X 0,Y 581.031,Z 664.443,A -85,B 0,C 180,E1 26515.916,E2 26515.916} C_VEL
LIN {X 0,Y 581.329,Z 605.048,A -85,B 0,C 180,E1 26515.027,E2 26515.027} C_VEL
LIN {X 0,Y 582.267,Z 398.476,A -85,B 0,C 180,E1 26511.988,E2 26511.988} C_VEL
LIN {X 0,Y 582.503,Z 316.324,A -85,B 0,C 180,E1 26510.736,E2 26510.736} C_VEL
LIN {X 0,Y 581.938,Z 310.616,A -85,B 0,C 180,E1 26510.558,E2 26510.558} C_VEL
LIN {X 0,Y 582.835,Z 248.418,A -85,B 0,C 180,E1 26507.608,E2 26507.608} C_VEL
LIN {X 0,Y 582.886,Z 240.392,A -85,B 0,C 180,E1 26507.212,E2 26507.212} C_VEL
LIN {X 0,Y 578.002,Z 231.524,A -85,B 0,C 180,E1 26506.309,E2 26506.309} C_VEL
LIN {X 0,Y 576.231,Z 228.144,A -85,B 0,C 180,E1 26505.953,E2 26505.953} C_VEL
LIN {X 0,Y 576.076,Z 227.316,A -85,B 0,C 180,E1 26505.754,E2 26505.754} C_VEL
LIN {X 0,Y 576.139,Z 227.265,A -85,B 0,C 180,E1 26502.596,E2 26502.596} C_VEL
LIN {X 0,Y 576.074,Z 227.282,A -85,B 0,C 180,E1 26499.567,E2 26499.567} C_VEL
LIN {X 0,Y 576.136,Z 227.284,A -85,B 0,C 180,E1 26496.365,E2 26496.365} C_VEL
LIN {X 0,Y 576.081,Z 227.284,A -85,B 0,C 180,E1 26493.38,E2 26493.38} C_VEL
LIN {X 0,Y 576.14,Z 227.28,A -85,B 0,C 180,E1 26490.202,E2 26490.202} C_VEL
LIN {X 0,Y 576.09,Z 227.283,A -85,B 0,C 180,E1 26487.159,E2 26487.159} C_VEL
LIN {X 0,Y 576.132,Z 227.28,A -85,B 0,C 180,E1 26483.96,E2 26483.96} C_VEL
LIN {X 0,Y 576.099,Z 227.281,A -85,B 0,C 180,E1 26480.949,E2 26480.949} C_VEL
LIN {X 0,Y 576.122,Z 227.279,A -85,B 0,C 180,E1 26477.675,E2 26477.675} C_VEL
LIN {X 0,Y 576.111,Z 227.281,A -85,B 0,C 180,E1 26474.678,E2 26474.678} C_VEL
LIN {X 0,Y 576.11,Z 227.278,A -85,B 0,C 180,E1 26471.31,E2 26471.31} C_VEL
LIN {X 0,Y 576.155,Z 227.282,A -85,B 0,C 180,E1 26468.181,E2 26468.181} C_VEL
LIN {X 0,Y 576.107,Z 227.277,A -85,B 0,C 180,E1 26464.979,E2 26464.979} C_VEL
LIN {X 0,Y 576.159,Z 227.275,A -85,B 0,C 180,E1 26461.79,E2 26461.79} C_VEL
LIN {X 0,Y 576.113,Z 227.28,A -85,B 0,C 180,E1 26458.608,E2 26458.608} C_VEL
LIN {X 0,Y 576.154,Z 227.274,A -85,B 0,C 180,E1 26455.322,E2 26455.322} C_VEL
LIN {X 0,Y 576.144,Z 227.282,A -85,B 0,C 180,E1 26452.02,E2 26452.02} C_VEL
LIN {X 0,Y 576.123,Z 227.277,A -85,B 0,C 180,E1 26448.684,E2 26448.684} C_VEL
LIN {X 0,Y 576.157,Z 227.278,A -85,B 0,C 180,E1 26445.529,E2 26445.529} C_VEL
LIN {X 0,Y 576.154,Z 227.278,A -85,B 0,C 180,E1 26443.353,E2 26443.353} C_VEL
LIN {X 0,Y 575.162,Z 227.398,A -85,B 0,C 180,E1 26442.587,E2 26442.587} C_VEL
LIN {X 0,Y 568.708,Z 228.198,A -85,B 0,C 180,E1 26440.437,E2 26440.437} C_VEL
LIN {X 0,Y 568.203,Z 228.265,A -85,B 0,C 180,E1 26439.877,E2 26439.877} C_VEL
LIN {X 0,Y 568.2,Z 228.262,A -85,B 0,C 180,E1 26436.567,E2 26436.567} C_VEL
LIN {X 0,Y 568.215,Z 228.269,A -85,B 0,C 180,E1 26433.34,E2 26433.34} C_VEL
LIN {X 0,Y 568.194,Z 228.262,A -85,B 0,C 180,E1 26430.017,E2 26430.017} C_VEL
LIN {X 0,Y 568.216,Z 228.261,A -85,B 0,C 180,E1 26426.702,E2 26426.702} C_VEL
LIN {X 0,Y 568.218,Z 228.271,A -85,B 0,C 180,E1 26423.254,E2 26423.254} C_VEL
LIN {X 0,Y 568.2,Z 228.261,A -85,B 0,C 180,E1 26419.907,E2 26419.907} C_VEL
LIN {X 0,Y 568.206,Z 228.262,A -85,B 0,C 180,E1 26416.665,E2 26416.665} C_VEL
LIN {X 0,Y 568.215,Z 228.271,A -85,B 0,C 180,E1 26413.336,E2 26413.336} C_VEL
LIN {X 0,Y 568.212,Z 228.263,A -85,B 0,C 180,E1 26409.897,E2 26409.897} C_VEL
LIN {X 0,Y 568.199,Z 228.267,A -85,B 0,C 180,E1 26406.623,E2 26406.623} C_VEL
LIN {X 0,Y 568.209,Z 228.266,A -85,B 0,C 180,E1 26403.421,E2 26403.421} C_VEL
LIN {X 0,Y 568.198,Z 228.263,A -85,B 0,C 180,E1 26400.218,E2 26400.218} C_VEL
LIN {X 0,Y 568.214,Z 228.268,A -85,B 0,C 180,E1 26396.858,E2 26396.858} C_VEL
LIN {X 0,Y 568.218,Z 228.263,A -85,B 0,C 180,E1 26393.543,E2 26393.543} C_VEL
LIN {X 0,Y 568.19,Z 228.269,A -85,B 0,C 180,E1 26390.284,E2 26390.284} C_VEL
LIN {X 0,Y 568.216,Z 228.256,A -85,B 0,C 180,E1 26386.985,E2 26386.985} C_VEL
LIN {X 0,Y 568.193,Z 228.267,A -85,B 0,C 180,E1 26383.744,E2 26383.744} C_VEL
LIN {X 0,Y 568.194,Z 228.273,A -85,B 0,C 180,E1 26380.341,E2 26380.341} C_VEL
LIN {X 0,Y 568.24,Z 228.51,A -85,B 0,C 180,E1 26379.419,E2 26379.419} C_VEL
LIN {X 0,Y 569.662,Z 231.937,A -85,B 0,C 180,E1 26379.034,E2 26379.034} C_VEL
LIN {X 0,Y 573.9,Z 241.56,A -85,B 0,C 180,E1 26378.088,E2 26378.088} C_VEL
LIN {X 0,Y 572.511,Z 294.851,A -85,B 0,C 180,E1 26374.86,E2 26374.86} C_VEL
LIN {X 0,Y 571.321,Z 350.191,A -85,B 0,C 180,E1 26371.606,E2 26371.606} C_VEL
LIN {X 0,Y 570.565,Z 410.338,A -85,B 0,C 180,E1 26368.244,E2 26368.244} C_VEL
LIN {X 0,Y 570.592,Z 418.248,A -85,B 0,C 180,E1 26367.839,E2 26367.839} C_VEL
LIN {X 0,Y 571.024,Z 425.521,A -85,B 0,C 180,E1 26367.721,E2 26367.721} C_VEL
LIN {X 0,Y 570.36,Z 628.317,A -85,B 0,C 180,E1 26365.017,E2 26365.017} C_VEL
LIN {X 0,Y 570.166,Z 647.355,A -85,B 0,C 180,E1 26364.57,E2 26364.57} C_VEL
LIN {X 0,Y 569.935,Z 665.417,A -85,B 0,C 180,E1 26363.959,E2 26363.959} C_VEL
LIN {X 0,Y 569.633,Z 683.499,A -85,B 0,C 180,E1 26363.146,E2 26363.146} C_VEL
LIN {X 0,Y 569.338,Z 700.47,A -85,B 0,C 180,E1 26362.179,E2 26362.179} C_VEL
LIN {X 0,Y 569.034,Z 716.506,A -85,B 0,C 180,E1 26361.055,E2 26361.055} C_VEL
LIN {X 0,Y 568.744,Z 731.605,A -85,B 0,C 180,E1 26359.774,E2 26359.774} C_VEL
LIN {X 0,Y 568.49,Z 745.709,A -85,B 0,C 180,E1 26358.332,E2 26358.332} C_VEL
LIN {X 0,Y 568.283,Z 758.34,A -85,B 0,C 180,E1 26356.779,E2 26356.779} C_VEL
LIN {X 0,Y 568.135,Z 768.887,A -85,B 0,C 180,E1 26355.217,E2 26355.217} C_VEL
LIN {X 0,Y 568.031,Z 778.21,A -85,B 0,C 180,E1 26353.538,E2 26353.538} C_VEL
LIN {X 0,Y 567.964,Z 786.202,A -85,B 0,C 180,E1 26351.74,E2 26351.74} C_VEL
LIN {X 0,Y 567.931,Z 792.396,A -85,B 0,C 180,E1 26349.923,E2 26349.923} C_VEL
LIN {X 0,Y 567.912,Z 796.895,A -85,B 0,C 180,E1 26348.086,E2 26348.086} C_VEL
LIN {X 0,Y 567.917,Z 799.736,A -85,B 0,C 180,E1 26346.225,E2 26346.225} C_VEL
LIN {X 0,Y 567.912,Z 800.921,A -85,B 0,C 180,E1 26344.337,E2 26344.337} C_VEL
LIN {X 0,Y 567.912,Z 800.401,A -85,B 0,C 180,E1 26342.418,E2 26342.418} C_VEL
LIN {X 0,Y 567.91,Z 798.257,A -85,B 0,C 180,E1 26340.582,E2 26340.582} C_VEL
LIN {X 0,Y 567.924,Z 794.376,A -85,B 0,C 180,E1 26338.712,E2 26338.712} C_VEL
LIN {X 0,Y 567.946,Z 788.994,A -85,B 0,C 180,E1 26336.926,E2 26336.926} C_VEL
LIN {X 0,Y 567.996,Z 781.7,A -85,B 0,C 180,E1 26335.105,E2 26335.105} C_VEL
LIN {X 0,Y 568.089,Z 772.884,A -85,B 0,C 180,E1 26333.371,E2 26333.371} C_VEL
LIN {X 0,Y 568.227,Z 762.407,A -85,B 0,C 180,E1 26331.7,E2 26331.7} C_VEL
LIN {X 0,Y 568.4,Z 750.95,A -85,B 0,C 180,E1 26330.188,E2 26330.188} C_VEL
LIN {X 0,Y 568.631,Z 737.927,A -85,B 0,C 180,E1 26328.749,E2 26328.749} C_VEL
LIN {X 0,Y 568.9,Z 723.52,A -85,B 0,C 180,E1 26327.42,E2 26327.42} C_VEL
LIN {X 0,Y 569.206,Z 707.654,A -85,B 0,C 180,E1 26326.206,E2 26326.206} C_VEL
LIN {X 0,Y 569.49,Z 691.239,A -85,B 0,C 180,E1 26325.177,E2 26325.177} C_VEL
LIN {X 0,Y 569.818,Z 673.432,A -85,B 0,C 180,E1 26324.284,E2 26324.284} C_VEL
LIN {X 0,Y 570.092,Z 654.822,A -85,B 0,C 180,E1 26323.568,E2 26323.568} C_VEL
LIN {X 0,Y 570.295,Z 635.853,A -85,B 0,C 180,E1 26323.047,E2 26323.047} C_VEL
LIN {X 0,Y 570.432,Z 616.046,A -85,B 0,C 180,E1 26322.706,E2 26322.706} C_VEL
LIN {X 0,Y 570.902,Z 420.762,A -85,B 0,C 180,E1 26320.119,E2 26320.119} C_VEL
LIN {X 0,Y 570.489,Z 416.683,A -85,B 0,C 180,E1 26320.015,E2 26320.015} C_VEL
LIN {X 0,Y 571.174,Z 359.647,A -85,B 0,C 180,E1 26316.837,E2 26316.837} C_VEL
LIN {X 0,Y 572.364,Z 309.13,A -85,B 0,C 180,E1 26313.866,E2 26313.866} C_VEL
LIN {X 0,Y 573.99,Z 254.136,A -85,B 0,C 180,E1 26310.515,E2 26310.515} C_VEL
LIN {X 0,Y 574.251,Z 241.972,A -85,B 0,C 180,E1 26309.75,E2 26309.75} C_VEL
LIN {X 0,Y 569.326,Z 231.562,A -85,B 0,C 180,E1 26308.649,E2 26308.649} C_VEL
LIN {X 0,Y 568.184,Z 228.607,A -85,B 0,C 180,E1 26308.31,E2 26308.31} C_VEL
LIN {X 0,Y 568.175,Z 228.263,A -85,B 0,C 180,E1 26307.569,E2 26307.569} C_VEL
LIN {X 0,Y 568.137,Z 228.269,A -85,B 0,C 180,E1 26304.318,E2 26304.318} C_VEL
LIN {X 0,Y 568.179,Z 228.267,A -85,B 0,C 180,E1 26301.362,E2 26301.362} C_VEL
LIN {X 0,Y 568.137,Z 228.274,A -85,B 0,C 180,E1 26298.138,E2 26298.138} C_VEL
LIN {X 0,Y 568.211,Z 228.272,A -85,B 0,C 180,E1 26294.978,E2 26294.978} C_VEL
LIN {X 0,Y 568.133,Z 228.273,A -85,B 0,C 180,E1 26291.779,E2 26291.779} C_VEL
LIN {X 0,Y 568.203,Z 228.271,A -85,B 0,C 180,E1 26288.602,E2 26288.602} C_VEL
LIN {X 0,Y 568.133,Z 228.273,A -85,B 0,C 180,E1 26285.554,E2 26285.554} C_VEL
LIN {X 0,Y 568.198,Z 228.271,A -85,B 0,C 180,E1 26282.42,E2 26282.42} C_VEL
LIN {X 0,Y 568.132,Z 228.271,A -85,B 0,C 180,E1 26279.395,E2 26279.395} C_VEL
LIN {X 0,Y 568.2,Z 228.273,A -85,B 0,C 180,E1 26276.267,E2 26276.267} C_VEL
LIN {X 0,Y 568.13,Z 228.272,A -85,B 0,C 180,E1 26273.228,E2 26273.228} C_VEL
LIN {X 0,Y 568.196,Z 228.274,A -85,B 0,C 180,E1 26270.069,E2 26270.069} C_VEL
LIN {X 0,Y 568.132,Z 228.273,A -85,B 0,C 180,E1 26266.981,E2 26266.981} C_VEL
LIN {X 0,Y 568.175,Z 228.273,A -85,B 0,C 180,E1 26263.751,E2 26263.751} C_VEL
LIN {X 0,Y 568.134,Z 228.273,A -85,B 0,C 180,E1 26260.786,E2 26260.786} C_VEL
LIN {X 0,Y 568.166,Z 228.271,A -85,B 0,C 180,E1 26257.498,E2 26257.498} C_VEL
LIN {X 0,Y 568.139,Z 228.273,A -85,B 0,C 180,E1 26254.527,E2 26254.527} C_VEL
LIN {X 0,Y 568.151,Z 228.274,A -85,B 0,C 180,E1 26251.171,E2 26251.171} C_VEL
LIN {X 0,Y 568.149,Z 228.274,A -85,B 0,C 180,E1 26248.209,E2 26248.209} C_VEL
LIN {X 0,Y 568.143,Z 228.275,A -85,B 0,C 180,E1 26244.867,E2 26244.867} C_VEL
LIN {X 0,Y 568.166,Z 228.276,A -85,B 0,C 180,E1 26241.852,E2 26241.852} C_VEL
LIN {X 0,Y 568.138,Z 228.277,A -85,B 0,C 180,E1 26238.563,E2 26238.563} C_VEL
LIN {X 0,Y 568.202,Z 228.27,A -85,B 0,C 180,E1 26235.403,E2 26235.403} C_VEL
LIN {X 0,Y 568.201,Z 228.507,A -85,B 0,C 180,E1 26234.879,E2 26234.879} C_VEL
LIN {X 0,Y 568.497,Z 229.799,A -85,B 0,C 180,E1 26234.707,E2 26234.707} C_VEL
LIN {X 0,Y 570.439,Z 232.958,A -85,B 0,C 180,E1 26234.346,E2 26234.346} C_VEL
LIN {X 0,Y 572.878,Z 237.381,A -85,B 0,C 180,E1 26233.878,E2 26233.878} C_VEL
LIN {X 0,Y 576.757,Z 244.853,A -85,B 0,C 180,E1 26233.127,E2 26233.127} C_VEL
LIN {X 0,Y 575.629,Z 306.562,A -85,B 0,C 180,E1 26230.158,E2 26230.158} C_VEL
LIN {X 0,Y 575.749,Z 313.629,A -85,B 0,C 180,E1 26229.858,E2 26229.858} C_VEL
LIN {X 0,Y 576.459,Z 320.971,A -85,B 0,C 180,E1 26229.683,E2 26229.683} C_VEL
LIN {X 0,Y 575.183,Z 532.31,A -85,B 0,C 180,E1 26226.501,E2 26226.501} C_VEL
LIN {X 0,Y 574.406,Z 662.872,A -85,B 0,C 180,E1 26224.56,E2 26224.56} C_VEL
LIN {X 0,Y 573.995,Z 686.687,A -85,B 0,C 180,E1 26224.019,E2 26224.019} C_VEL
LIN {X 0,Y 573.615,Z 708.471,A -85,B 0,C 180,E1 26223.339,E2 26223.339} C_VEL
LIN {X 0,Y 573.02,Z 730.72,A -85,B 0,C 180,E1 26222.448,E2 26222.448} C_VEL
LIN {X 0,Y 572.503,Z 751.817,A -85,B 0,C 180,E1 26221.419,E2 26221.419} C_VEL
LIN {X 0,Y 571.824,Z 772.958,A -85,B 0,C 180,E1 26220.178,E2 26220.178} C_VEL
LIN {X 0,Y 571.196,Z 794.124,A -85,B 0,C 180,E1 26218.72,E2 26218.72} C_VEL
LIN {X 0,Y 570.578,Z 812.928,A -85,B 0,C 180,E1 26217.216,E2 26217.216} C_VEL
LIN {X 0,Y 570.014,Z 831.472,A -85,B 0,C 180,E1 26215.506,E2 26215.506} C_VEL
LIN {X 0,Y 569.517,Z 848.629,A -85,B 0,C 180,E1 26213.704,E2 26213.704} C_VEL
LIN {X 0,Y 569.056,Z 864.704,A -85,B 0,C 180,E1 26211.76,E2 26211.76} C_VEL
LIN {X 0,Y 568.704,Z 879.343,A -85,B 0,C 180,E1 26209.727,E2 26209.727} C_VEL
LIN {X 0,Y 568.448,Z 892.016,A -85,B 0,C 180,E1 26207.714,E2 26207.714} C_VEL
LIN {X 0,Y 568.237,Z 903.324,A -85,B 0,C 180,E1 26205.616,E2 26205.616} C_VEL
LIN {X 0,Y 568.102,Z 913.461,A -85,B 0,C 180,E1 26203.432,E2 26203.432} C_VEL
LIN {X 0,Y 567.995,Z 921.7,A -85,B 0,C 180,E1 26201.267,E2 26201.267} C_VEL
LIN {X 0,Y 567.953,Z 928.739,A -85,B 0,C 180,E1 26199.027,E2 26199.027} C_VEL
LIN {X 0,Y 567.92,Z 934.049,A -85,B 0,C 180,E1 26196.773,E2 26196.773} C_VEL
LIN {X 0,Y 567.9,Z 937.915,A -85,B 0,C 180,E1 26194.543,E2 26194.543} C_VEL
LIN {X 0,Y 567.904,Z 940.123,A -85,B 0,C 180,E1 26192.32,E2 26192.32} C_VEL
LIN {X 0,Y 567.91,Z 940.984,A -85,B 0,C 180,E1 26190.1,E2 26190.1} C_VEL
LIN {X 0,Y 567.906,Z 940.189,A -85,B 0,C 180,E1 26187.779,E2 26187.779} C_VEL
LIN {X 0,Y 567.902,Z 938.048,A -85,B 0,C 180,E1 26185.556,E2 26185.556} C_VEL
LIN {X 0,Y 567.922,Z 934.252,A -85,B 0,C 180,E1 26183.326,E2 26183.326} C_VEL
LIN {X 0,Y 567.934,Z 929.293,A -85,B 0,C 180,E1 26181.189,E2 26181.189} C_VEL
LIN {X 0,Y 567.982,Z 922.404,A -85,B 0,C 180,E1 26178.937,E2 26178.937} C_VEL
LIN {X 0,Y 568.079,Z 914.695,A -85,B 0,C 180,E1 26176.876,E2 26176.876} C_VEL
LIN {X 0,Y 568.216,Z 904.356,A -85,B 0,C 180,E1 26174.59,E2 26174.59} C_VEL
LIN {X 0,Y 568.429,Z 892.897,A -85,B 0,C 180,E1 26172.433,E2 26172.433} C_VEL
LIN {X 0,Y 568.68,Z 880.037,A -85,B 0,C 180,E1 26170.377,E2 26170.377} C_VEL
LIN {X 0,Y 569.036,Z 865.532,A -85,B 0,C 180,E1 26168.346,E2 26168.346} C_VEL
LIN {X 0,Y 569.46,Z 850.47,A -85,B 0,C 180,E1 26166.511,E2 26166.511} C_VEL
LIN {X 0,Y 569.952,Z 833.108,A -85,B 0,C 180,E1 26164.656,E2 26164.656} C_VEL
LIN {X 0,Y 570.54,Z 814.884,A -85,B 0,C 180,E1 26162.949,E2 26162.949} C_VEL
LIN {X 0,Y 571.141,Z 795.6,A -85,B 0,C 180,E1 26161.392,E2 26161.392} C_VEL
LIN {X 0,Y 571.765,Z 774.701,A -85,B 0,C 180,E1 26159.932,E2 26159.932} C_VEL
LIN {X 0,Y 572.401,Z 754.818,A -85,B 0,C 180,E1 26158.748,E2 26158.748} C_VEL
LIN {X 0,Y 572.973,Z 732.427,A -85,B 0,C 180,E1 26157.629,E2 26157.629} C_VEL
LIN {X 0,Y 573.583,Z 710.347,A -85,B 0,C 180,E1 26156.727,E2 26156.727} C_VEL
LIN {X 0,Y 573.983,Z 687.839,A -85,B 0,C 180,E1 26156.014,E2 26156.014} C_VEL
LIN {X 0,Y 574.392,Z 664.979,A -85,B 0,C 180,E1 26155.476,E2 26155.476} C_VEL
LIN {X 0,Y 574.748,Z 609.612,A -85,B 0,C 180,E1 26154.636,E2 26154.636} C_VEL
LIN {X 0,Y 575.931,Z 403.048,A -85,B 0,C 180,E1 26151.565,E2 26151.565} C_VEL
LIN {X 0,Y 576.294,Z 317.732,A -85,B 0,C 180,E1 26150.252,E2 26150.252} C_VEL
LIN {X 0,Y 575.558,Z 310.615,A -85,B 0,C 180,E1 26150.033,E2 26150.033} C_VEL
LIN {X 0,Y 576.692,Z 248.418,A -85,B 0,C 180,E1 26147.048,E2 26147.048} C_VEL
LIN {X 0,Y 576.67,Z 244.483,A -85,B 0,C 180,E1 26146.846,E2 26146.846} C_VEL
LIN {X 0,Y 572.338,Z 236.686,A -85,B 0,C 180,E1 26146.034,E2 26146.034} C_VEL
LIN {X 0,Y 569.905,Z 232.366,A -85,B 0,C 180,E1 26145.571,E2 26145.571} C_VEL
LIN {X 0,Y 568.242,Z 228.79,A -85,B 0,C 180,E1 26145.184,E2 26145.184} C_VEL
LIN {X 0,Y 568.203,Z 228.274,A -85,B 0,C 180,E1 26144.833,E2 26144.833} C_VEL
LIN {X 0,Y 568.133,Z 228.272,A -85,B 0,C 180,E1 26141.701,E2 26141.701} C_VEL
LIN {X 0,Y 568.209,Z 228.272,A -85,B 0,C 180,E1 26138.62,E2 26138.62} C_VEL
LIN {X 0,Y 568.14,Z 228.274,A -85,B 0,C 180,E1 26135.504,E2 26135.504} C_VEL
LIN {X 0,Y 568.209,Z 228.267,A -85,B 0,C 180,E1 26132.34,E2 26132.34} C_VEL
LIN {X 0,Y 568.147,Z 228.271,A -85,B 0,C 180,E1 26129.291,E2 26129.291} C_VEL
LIN {X 0,Y 568.202,Z 228.266,A -85,B 0,C 180,E1 26126.099,E2 26126.099} C_VEL
LIN {X 0,Y 568.159,Z 228.272,A -85,B 0,C 180,E1 26122.997,E2 26122.997} C_VEL
LIN {X 0,Y 568.174,Z 228.268,A -85,B 0,C 180,E1 26119.641,E2 26119.641} C_VEL
LIN {X 0,Y 568.186,Z 228.271,A -85,B 0,C 180,E1 26116.564,E2 26116.564} C_VEL
LIN {X 0,Y 568.167,Z 228.268,A -85,B 0,C 180,E1 26113.301,E2 26113.301} C_VEL
LIN {X 0,Y 568.217,Z 228.267,A -85,B 0,C 180,E1 26110.135,E2 26110.135} C_VEL
LIN {X 0,Y 568.166,Z 228.268,A -85,B 0,C 180,E1 26106.975,E2 26106.975} C_VEL
LIN {X 0,Y 568.223,Z 228.267,A -85,B 0,C 180,E1 26103.733,E2 26103.733} C_VEL
LIN {X 0,Y 568.177,Z 228.264,A -85,B 0,C 180,E1 26100.505,E2 26100.505} C_VEL
LIN {X 0,Y 568.195,Z 228.263,A -85,B 0,C 180,E1 26097.176,E2 26097.176} C_VEL
LIN {X 0,Y 568.216,Z 228.271,A -85,B 0,C 180,E1 26093.94,E2 26093.94} C_VEL
LIN {X 0,Y 568.181,Z 228.262,A -85,B 0,C 180,E1 26090.683,E2 26090.683} C_VEL
LIN {X 0,Y 568.218,Z 228.265,A -85,B 0,C 180,E1 26087.501,E2 26087.501} C_VEL
LIN {X 0,Y 568.185,Z 228.267,A -85,B 0,C 180,E1 26084.277,E2 26084.277} C_VEL
LIN {X 0,Y 568.217,Z 228.257,A -85,B 0,C 180,E1 26081.003,E2 26081.003} C_VEL
LIN {X 0,Y 568.203,Z 228.265,A -85,B 0,C 180,E1 26079.877,E2 26079.877} C_VEL
LIN {X 0,Y 567.252,Z 228.391,A -85,B 0,C 180,E1 26079.1,E2 26079.1} C_VEL
LIN {X 0,Y 560.704,Z 229.198,A -85,B 0,C 180,E1 26076.863,E2 26076.863} C_VEL
LIN {X 0,Y 560.253,Z 229.253,A -85,B 0,C 180,E1 26076.351,E2 26076.351} C_VEL
LIN {X 0,Y 560.275,Z 229.255,A -85,B 0,C 180,E1 26073.046,E2 26073.046} C_VEL
LIN {X 0,Y 560.266,Z 229.252,A -85,B 0,C 180,E1 26069.742,E2 26069.742} C_VEL
LIN {X 0,Y 560.265,Z 229.251,A -85,B 0,C 180,E1 26066.289,E2 26066.289} C_VEL
LIN {X 0,Y 560.271,Z 229.257,A -85,B 0,C 180,E1 26063.03,E2 26063.03} C_VEL
LIN {X 0,Y 560.26,Z 229.251,A -85,B 0,C 180,E1 26059.757,E2 26059.757} C_VEL
LIN {X 0,Y 560.276,Z 229.248,A -85,B 0,C 180,E1 26056.431,E2 26056.431} C_VEL
LIN {X 0,Y 560.271,Z 229.256,A -85,B 0,C 180,E1 26052.973,E2 26052.973} C_VEL
LIN {X 0,Y 560.269,Z 229.254,A -85,B 0,C 180,E1 26049.71,E2 26049.71} C_VEL
LIN {X 0,Y 560.262,Z 229.254,A -85,B 0,C 180,E1 26046.404,E2 26046.404} C_VEL
LIN {X 0,Y 560.277,Z 229.255,A -85,B 0,C 180,E1 26043.099,E2 26043.099} C_VEL
LIN {X 0,Y 560.277,Z 229.25,A -85,B 0,C 180,E1 26039.649,E2 26039.649} C_VEL
LIN {X 0,Y 560.255,Z 229.255,A -85,B 0,C 180,E1 26036.378,E2 26036.378} C_VEL
LIN {X 0,Y 560.275,Z 229.25,A -85,B 0,C 180,E1 26033.118,E2 26033.118} C_VEL
LIN {X 0,Y 560.262,Z 229.254,A -85,B 0,C 180,E1 26029.822,E2 26029.822} C_VEL
LIN {X 0,Y 560.251,Z 229.242,A -85,B 0,C 180,E1 26026.379,E2 26026.379} C_VEL
LIN {X 0,Y 560.278,Z 229.244,A -85,B 0,C 180,E1 26023.1,E2 26023.1} C_VEL
LIN {X 0,Y 560.275,Z 229.489,A -85,B 0,C 180,E1 26020.021,E2 26020.021} C_VEL
LIN {X 0,Y 561.017,Z 231.812,A -85,B 0,C 180,E1 26019.749,E2 26019.749} C_VEL
LIN {X 0,Y 565.82,Z 242.027,A -85,B 0,C 180,E1 26018.691,E2 26018.691} C_VEL
LIN {X 0,Y 567.158,Z 245.47,A -85,B 0,C 180,E1 26018.364,E2 26018.364} C_VEL
LIN {X 0,Y 565.568,Z 299.239,A -85,B 0,C 180,E1 26015.072,E2 26015.072} C_VEL
LIN {X 0,Y 564.196,Z 353.819,A -85,B 0,C 180,E1 26011.829,E2 26011.829} C_VEL
LIN {X 0,Y 563.243,Z 403.223,A -85,B 0,C 180,E1 26008.984,E2 26008.984} C_VEL
LIN {X 0,Y 563.154,Z 418.186,A -85,B 0,C 180,E1 26008.176,E2 26008.176} C_VEL
LIN {X 0,Y 563.702,Z 425.886,A -85,B 0,C 180,E1 26008.044,E2 26008.044} C_VEL
LIN {X 0,Y 562.894,Z 628.284,A -85,B 0,C 180,E1 26005.31,E2 26005.31} C_VEL
LIN {X 0,Y 562.661,Z 647.334,A -85,B 0,C 180,E1 26004.859,E2 26004.859} C_VEL
LIN {X 0,Y 562.375,Z 665.614,A -85,B 0,C 180,E1 26004.231,E2 26004.231} C_VEL
LIN {X 0,Y 562.04,Z 682.608,A -85,B 0,C 180,E1 26003.464,E2 26003.464} C_VEL
LIN {X 0,Y 561.67,Z 699.764,A -85,B 0,C 180,E1 26002.483,E2 26002.483} C_VEL
LIN {X 0,Y 561.303,Z 715.903,A -85,B 0,C 180,E1 26001.346,E2 26001.346} C_VEL
LIN {X 0,Y 560.948,Z 731.127,A -85,B 0,C 180,E1 26000.045,E2 26000.045} C_VEL
LIN {X 0,Y 560.634,Z 745.31,A -85,B 0,C 180,E1 25998.583,E2 25998.583} C_VEL
LIN {X 0,Y 560.38,Z 758.001,A -85,B 0,C 180,E1 25997.009,E2 25997.009} C_VEL
LIN {X 0,Y 560.184,Z 769.248,A -85,B 0,C 180,E1 25995.319,E2 25995.319} C_VEL
LIN {X 0,Y 560.06,Z 778.501,A -85,B 0,C 180,E1 25993.617,E2 25993.617} C_VEL
LIN {X 0,Y 559.974,Z 786.431,A -85,B 0,C 180,E1 25991.793,E2 25991.793} C_VEL
LIN {X 0,Y 559.934,Z 792.64,A -85,B 0,C 180,E1 25989.926,E2 25989.926} C_VEL
LIN {X 0,Y 559.913,Z 797.01,A -85,B 0,C 180,E1 25988.087,E2 25988.087} C_VEL
LIN {X 0,Y 559.915,Z 799.799,A -85,B 0,C 180,E1 25986.2,E2 25986.2} C_VEL
LIN {X 0,Y 559.912,Z 800.934,A -85,B 0,C 180,E1 25984.284,E2 25984.284} C_VEL
LIN {X 0,Y 559.912,Z 800.361,A -85,B 0,C 180,E1 25982.337,E2 25982.337} C_VEL
LIN {X 0,Y 559.913,Z 798.074,A -85,B 0,C 180,E1 25980.417,E2 25980.417} C_VEL
LIN {X 0,Y 559.928,Z 794.22,A -85,B 0,C 180,E1 25978.574,E2 25978.574} C_VEL
LIN {X 0,Y 559.955,Z 788.51,A -85,B 0,C 180,E1 25976.684,E2 25976.684} C_VEL
LIN {X 0,Y 560.031,Z 781.149,A -85,B 0,C 180,E1 25974.853,E2 25974.853} C_VEL
LIN {X 0,Y 560.142,Z 772.217,A -85,B 0,C 180,E1 25973.099,E2 25973.099} C_VEL
LIN {X 0,Y 560.316,Z 761.609,A -85,B 0,C 180,E1 25971.405,E2 25971.405} C_VEL
LIN {X 0,Y 560.554,Z 749.284,A -85,B 0,C 180,E1 25969.784,E2 25969.784} C_VEL
LIN {X 0,Y 560.846,Z 735.903,A -85,B 0,C 180,E1 25968.322,E2 25968.322} C_VEL
LIN {X 0,Y 561.181,Z 721.023,A -85,B 0,C 180,E1 25966.971,E2 25966.971} C_VEL
LIN {X 0,Y 561.541,Z 705.466,A -85,B 0,C 180,E1 25965.801,E2 25965.801} C_VEL
LIN {X 0,Y 561.898,Z 688.671,A -85,B 0,C 180,E1 25964.768,E2 25964.768} C_VEL
LIN {X 0,Y 562.261,Z 671.169,A -85,B 0,C 180,E1 25963.909,E2 25963.909} C_VEL
LIN {X 0,Y 562.578,Z 652.907,A -85,B 0,C 180,E1 25963.223,E2 25963.223} C_VEL
LIN {X 0,Y 562.823,Z 634.309,A -85,B 0,C 180,E1 25962.723,E2 25962.723} C_VEL
LIN {X 0,Y 562.984,Z 613.277,A -85,B 0,C 180,E1 25962.374,E2 25962.374} C_VEL
LIN {X 0,Y 563.57,Z 421.602,A -85,B 0,C 180,E1 25959.801,E2 25959.801} C_VEL
LIN {X 0,Y 563.05,Z 416.544,A -85,B 0,C 180,E1 25959.671,E2 25959.671} C_VEL
LIN {X 0,Y 563.872,Z 369.868,A -85,B 0,C 180,E1 25957.013,E2 25957.013} C_VEL
LIN {X 0,Y 565.53,Z 311.856,A -85,B 0,C 180,E1 25953.538,E2 25953.538} C_VEL
LIN {X 0,Y 567.363,Z 256.781,A -85,B 0,C 180,E1 25950.148,E2 25950.148} C_VEL
LIN {X 0,Y 567.638,Z 245.584,A -85,B 0,C 180,E1 25949.435,E2 25949.435} C_VEL
LIN {X 0,Y 561.511,Z 232.754,A -85,B 0,C 180,E1 25948.04,E2 25948.04} C_VEL
LIN {X 0,Y 560.277,Z 229.605,A -85,B 0,C 180,E1 25947.673,E2 25947.673} C_VEL
LIN {X 0,Y 560.259,Z 229.247,A -85,B 0,C 180,E1 25947.063,E2 25947.063} C_VEL
LIN {X 0,Y 560.2,Z 229.258,A -85,B 0,C 180,E1 25943.964,E2 25943.964} C_VEL
LIN {X 0,Y 560.233,Z 229.258,A -85,B 0,C 180,E1 25940.693,E2 25940.693} C_VEL
LIN {X 0,Y 560.204,Z 229.263,A -85,B 0,C 180,E1 25937.662,E2 25937.662} C_VEL
LIN {X 0,Y 560.208,Z 229.263,A -85,B 0,C 180,E1 25934.258,E2 25934.258} C_VEL
LIN {X 0,Y 560.225,Z 229.262,A -85,B 0,C 180,E1 25931.217,E2 25931.217} C_VEL
LIN {X 0,Y 560.199,Z 229.26,A -85,B 0,C 180,E1 25927.899,E2 25927.899} C_VEL
LIN {X 0,Y 560.238,Z 229.261,A -85,B 0,C 180,E1 25924.914,E2 25924.914} C_VEL
LIN {X 0,Y 560.196,Z 229.262,A -85,B 0,C 180,E1 25921.738,E2 25921.738} C_VEL
LIN {X 0,Y 560.235,Z 229.259,A -85,B 0,C 180,E1 25918.772,E2 25918.772} C_VEL
LIN {X 0,Y 560.194,Z 229.263,A -85,B 0,C 180,E1 25915.495,E2 25915.495} C_VEL
LIN {X 0,Y 560.274,Z 229.261,A -85,B 0,C 180,E1 25912.308,E2 25912.308} C_VEL
LIN {X 0,Y 560.193,Z 229.263,A -85,B 0,C 180,E1 25909.094,E2 25909.094} C_VEL
LIN {X 0,Y 560.24,Z 229.26,A -85,B 0,C 180,E1 25905.847,E2 25905.847} C_VEL
LIN {X 0,Y 560.195,Z 229.262,A -85,B 0,C 180,E1 25902.872,E2 25902.872} C_VEL
LIN {X 0,Y 560.235,Z 229.261,A -85,B 0,C 180,E1 25899.634,E2 25899.634} C_VEL
LIN {X 0,Y 560.197,Z 229.26,A -85,B 0,C 180,E1 25896.657,E2 25896.657} C_VEL
LIN {X 0,Y 560.228,Z 229.263,A -85,B 0,C 180,E1 25893.386,E2 25893.386} C_VEL
LIN {X 0,Y 560.204,Z 229.263,A -85,B 0,C 180,E1 25890.363,E2 25890.363} C_VEL
LIN {X 0,Y 560.202,Z 229.264,A -85,B 0,C 180,E1 25886.896,E2 25886.896} C_VEL
LIN {X 0,Y 560.244,Z 229.263,A -85,B 0,C 180,E1 25883.77,E2 25883.77} C_VEL
LIN {X 0,Y 560.197,Z 229.264,A -85,B 0,C 180,E1 25880.55,E2 25880.55} C_VEL
LIN {X 0,Y 560.262,Z 229.255,A -85,B 0,C 180,E1 25877.439,E2 25877.439} C_VEL
LIN {X 0,Y 560.277,Z 229.485,A -85,B 0,C 180,E1 25875.545,E2 25875.545} C_VEL
LIN {X 0,Y 560.749,Z 231.166,A -85,B 0,C 180,E1 25875.351,E2 25875.351} C_VEL
LIN {X 0,Y 564.788,Z 238.193,A -85,B 0,C 180,E1 25874.629,E2 25874.629} C_VEL
LIN {X 0,Y 570.585,Z 248.622,A -85,B 0,C 180,E1 25873.515,E2 25873.515} C_VEL
LIN {X 0,Y 569.255,Z 309.333,A -85,B 0,C 180,E1 25870.564,E2 25870.564} C_VEL
LIN {X 0,Y 569.503,Z 314.347,A -85,B 0,C 180,E1 25870.373,E2 25870.373} C_VEL
LIN {X 0,Y 570.289,Z 322.243,A -85,B 0,C 180,E1 25870.178,E2 25870.178} C_VEL
LIN {X 0,Y 568.742,Z 533.455,A -85,B 0,C 180,E1 25866.965,E2 25866.965} C_VEL
LIN {X 0,Y 567.807,Z 663.087,A -85,B 0,C 180,E1 25865.016,E2 25865.016} C_VEL
LIN {X 0,Y 567.322,Z 686.816,A -85,B 0,C 180,E1 25864.471,E2 25864.471} C_VEL
LIN {X 0,Y 566.847,Z 708.906,A -85,B 0,C 180,E1 25863.775,E2 25863.775} C_VEL
LIN {X 0,Y 566.165,Z 730.724,A -85,B 0,C 180,E1 25862.89,E2 25862.89} C_VEL
LIN {X 0,Y 565.505,Z 751.818,A -85,B 0,C 180,E1 25861.853,E2 25861.853} C_VEL
LIN {X 0,Y 564.721,Z 772.872,A -85,B 0,C 180,E1 25860.603,E2 25860.603} C_VEL
LIN {X 0,Y 563.962,Z 793.426,A -85,B 0,C 180,E1 25859.178,E2 25859.178} C_VEL
LIN {X 0,Y 563.248,Z 811.607,A -85,B 0,C 180,E1 25857.715,E2 25857.715} C_VEL
LIN {X 0,Y 562.522,Z 830.973,A -85,B 0,C 180,E1 25855.922,E2 25855.922} C_VEL
LIN {X 0,Y 561.905,Z 848.174,A -85,B 0,C 180,E1 25854.1,E2 25854.1} C_VEL
LIN {X 0,Y 561.364,Z 864.092,A -85,B 0,C 180,E1 25852.153,E2 25852.153} C_VEL
LIN {X 0,Y 560.904,Z 879.345,A -85,B 0,C 180,E1 25850.013,E2 25850.013} C_VEL
LIN {X 0,Y 560.562,Z 892.649,A -85,B 0,C 180,E1 25847.865,E2 25847.865} C_VEL
LIN {X 0,Y 560.306,Z 903.846,A -85,B 0,C 180,E1 25845.737,E2 25845.737} C_VEL
LIN {X 0,Y 560.14,Z 913.886,A -85,B 0,C 180,E1 25843.522,E2 25843.522} C_VEL
LIN {X 0,Y 560.016,Z 922.057,A -85,B 0,C 180,E1 25841.325,E2 25841.325} C_VEL
LIN {X 0,Y 559.96,Z 929.043,A -85,B 0,C 180,E1 25839.039,E2 25839.039} C_VEL
LIN {X 0,Y 559.922,Z 934.081,A -85,B 0,C 180,E1 25836.855,E2 25836.855} C_VEL
LIN {X 0,Y 559.9,Z 937.915,A -85,B 0,C 180,E1 25834.608,E2 25834.608} C_VEL
LIN {X 0,Y 559.905,Z 940.123,A -85,B 0,C 180,E1 25832.353,E2 25832.353} C_VEL
LIN {X 0,Y 559.91,Z 940.984,A -85,B 0,C 180,E1 25830.101,E2 25830.101} C_VEL
LIN {X 0,Y 559.906,Z 940.189,A -85,B 0,C 180,E1 25827.747,E2 25827.747} C_VEL
LIN {X 0,Y 559.901,Z 938.048,A -85,B 0,C 180,E1 25825.492,E2 25825.492} C_VEL
LIN {X 0,Y 559.922,Z 934.252,A -85,B 0,C 180,E1 25823.231,E2 25823.231} C_VEL
LIN {X 0,Y 559.948,Z 929.293,A -85,B 0,C 180,E1 25821.062,E2 25821.062} C_VEL
LIN {X 0,Y 560.008,Z 922.405,A -85,B 0,C 180,E1 25818.777,E2 25818.777} C_VEL
LIN {X 0,Y 560.131,Z 914.287,A -85,B 0,C 180,E1 25816.581,E2 25816.581} C_VEL
LIN {X 0,Y 560.295,Z 904.358,A -85,B 0,C 180,E1 25814.367,E2 25814.367} C_VEL
LIN {X 0,Y 560.547,Z 893.234,A -85,B 0,C 180,E1 25812.24,E2 25812.24} C_VEL
LIN {X 0,Y 560.88,Z 880.039,A -85,B 0,C 180,E1 25810.093,E2 25810.093} C_VEL
LIN {X 0,Y 561.311,Z 865.53,A -85,B 0,C 180,E1 25808.032,E2 25808.032} C_VEL
LIN {X 0,Y 561.835,Z 850.006,A -85,B 0,C 180,E1 25806.116,E2 25806.116} C_VEL
LIN {X 0,Y 562.458,Z 832.667,A -85,B 0,C 180,E1 25804.248,E2 25804.248} C_VEL
LIN {X 0,Y 563.12,Z 815.26,A -85,B 0,C 180,E1 25802.596,E2 25802.596} C_VEL
LIN {X 0,Y 563.845,Z 796.33,A -85,B 0,C 180,E1 25801.045,E2 25801.045} C_VEL
LIN {X 0,Y 564.61,Z 775.593,A -85,B 0,C 180,E1 25799.57,E2 25799.57} C_VEL
LIN {X 0,Y 565.355,Z 755.819,A -85,B 0,C 180,E1 25798.373,E2 25798.373} C_VEL
LIN {X 0,Y 566.073,Z 733.183,A -85,B 0,C 180,E1 25797.221,E2 25797.221} C_VEL
LIN {X 0,Y 566.733,Z 712.491,A -85,B 0,C 180,E1 25796.359,E2 25796.359} C_VEL
LIN {X 0,Y 567.279,Z 689.327,A -85,B 0,C 180,E1 25795.6,E2 25795.6} C_VEL
LIN {X 0,Y 567.742,Z 667.267,A -85,B 0,C 180,E1 25795.061,E2 25795.061} C_VEL
LIN {X 0,Y 568.085,Z 630.877,A -85,B 0,C 180,E1 25794.482,E2 25794.482} C_VEL
LIN {X 0,Y 569.511,Z 423.719,A -85,B 0,C 180,E1 25791.378,E2 25791.378} C_VEL
LIN {X 0,Y 570.127,Z 319.136,A -85,B 0,C 180,E1 25789.758,E2 25789.758} C_VEL
LIN {X 0,Y 569.22,Z 310.996,A -85,B 0,C 180,E1 25789.516,E2 25789.516} C_VEL
LIN {X 0,Y 570.589,Z 249.049,A -85,B 0,C 180,E1 25786.507,E2 25786.507} C_VEL
LIN {X 0,Y 568.461,Z 244.694,A -85,B 0,C 180,E1 25786.076,E2 25786.076} C_VEL
LIN {X 0,Y 562.831,Z 234.612,A -85,B 0,C 180,E1 25784.995,E2 25784.995} C_VEL
LIN {X 0,Y 560.53,Z 230.562,A -85,B 0,C 180,E1 25784.581,E2 25784.581} C_VEL
LIN {X 0,Y 560.247,Z 229.376,A -85,B 0,C 180,E1 25784.394,E2 25784.394} C_VEL
LIN {X 0,Y 560.205,Z 229.261,A -85,B 0,C 180,E1 25781.329,E2 25781.329} C_VEL
LIN {X 0,Y 560.206,Z 229.262,A -85,B 0,C 180,E1 25777.877,E2 25777.877} C_VEL
LIN {X 0,Y 560.245,Z 229.26,A -85,B 0,C 180,E1 25774.819,E2 25774.819} C_VEL
LIN {X 0,Y 560.207,Z 229.259,A -85,B 0,C 180,E1 25771.64,E2 25771.64} C_VEL
LIN {X 0,Y 560.265,Z 229.257,A -85,B 0,C 180,E1 25768.573,E2 25768.573} C_VEL
LIN {X 0,Y 560.211,Z 229.257,A -85,B 0,C 180,E1 25765.363,E2 25765.363} C_VEL
LIN {X 0,Y 560.283,Z 229.255,A -85,B 0,C 180,E1 25762.151,E2 25762.151} C_VEL
LIN {X 0,Y 560.222,Z 229.259,A -85,B 0,C 180,E1 25758.928,E2 25758.928} C_VEL
LIN {X 0,Y 560.238,Z 229.255,A -85,B 0,C 180,E1 25755.528,E2 25755.528} C_VEL
LIN {X 0,Y 560.25,Z 229.26,A -85,B 0,C 180,E1 25752.471,E2 25752.471} C_VEL
LIN {X 0,Y 560.229,Z 229.256,A -85,B 0,C 180,E1 25749.14,E2 25749.14} C_VEL
LIN {X 0,Y 560.285,Z 229.253,A -85,B 0,C 180,E1 25745.941,E2 25745.941} C_VEL
LIN {X 0,Y 560.233,Z 229.259,A -85,B 0,C 180,E1 25742.66,E2 25742.66} C_VEL
LIN {X 0,Y 560.272,Z 229.254,A -85,B 0,C 180,E1 25739.387,E2 25739.387} C_VEL
LIN {X 0,Y 560.263,Z 229.255,A -85,B 0,C 180,E1 25736.112,E2 25736.112} C_VEL
LIN {X 0,Y 560.244,Z 229.255,A -85,B 0,C 180,E1 25732.824,E2 25732.824} C_VEL
LIN {X 0,Y 560.281,Z 229.258,A -85,B 0,C 180,E1 25729.617,E2 25729.617} C_VEL
LIN {X 0,Y 560.245,Z 229.254,A -85,B 0,C 180,E1 25726.375,E2 25726.375} C_VEL
LIN {X 0,Y 560.28,Z 229.252,A -85,B 0,C 180,E1 25723.045,E2 25723.045} C_VEL
LIN {X 0,Y 560.28,Z 229.256,A -85,B 0,C 180,E1 25719.636,E2 25719.636} C_VEL
LIN {X 0,Y 560.253,Z 229.253,A -85,B 0,C 180,E1 25716.351,E2 25716.351} C_VEL
LIN {X 0,Y 559.256,Z 229.381,A -85,B 0,C 180,E1 25715.564,E2 25715.564} C_VEL
LIN {X 0,Y 552.865,Z 230.182,A -85,B 0,C 180,E1 25713.352,E2 25713.352} C_VEL
LIN {X 0,Y 552.34,Z 230.241,A -85,B 0,C 180,E1 25712.776,E2 25712.776} C_VEL
LIN {X 0,Y 552.342,Z 230.244,A -85,B 0,C 180,E1 25709.425,E2 25709.425} C_VEL
LIN {X 0,Y 552.32,Z 230.243,A -85,B 0,C 180,E1 25706.009,E2 25706.009} C_VEL
LIN {X 0,Y 552.337,Z 230.241,A -85,B 0,C 180,E1 25702.627,E2 25702.627} C_VEL
LIN {X 0,Y 552.338,Z 230.248,A -85,B 0,C 180,E1 25699.173,E2 25699.173} C_VEL
LIN {X 0,Y 552.326,Z 230.24,A -85,B 0,C 180,E1 25695.797,E2 25695.797} C_VEL
LIN {X 0,Y 552.33,Z 230.24,A -85,B 0,C 180,E1 25692.473,E2 25692.473} C_VEL
LIN {X 0,Y 552.339,Z 230.248,A -85,B 0,C 180,E1 25689.048,E2 25689.048} C_VEL
LIN {X 0,Y 552.333,Z 230.243,A -85,B 0,C 180,E1 25685.631,E2 25685.631} C_VEL
LIN {X 0,Y 552.322,Z 230.244,A -85,B 0,C 180,E1 25682.279,E2 25682.279} C_VEL
LIN {X 0,Y 552.335,Z 230.246,A -85,B 0,C 180,E1 25678.904,E2 25678.904} C_VEL
LIN {X 0,Y 552.339,Z 230.24,A -85,B 0,C 180,E1 25675.521,E2 25675.521} C_VEL
LIN {X 0,Y 552.309,Z 230.225,A -85,B 0,C 180,E1 25672.233,E2 25672.233} C_VEL
LIN {X 0,Y 552.34,Z 230.25,A -85,B 0,C 180,E1 25668.908,E2 25668.908} C_VEL
LIN {X 0,Y 552.333,Z 230.235,A -85,B 0,C 180,E1 25665.541,E2 25665.541} C_VEL
LIN {X 0,Y 552.304,Z 230.223,A -85,B 0,C 180,E1 25662.159,E2 25662.159} C_VEL
LIN {X 0,Y 552.366,Z 230.46,A -85,B 0,C 180,E1 25660.641,E2 25660.641} C_VEL
LIN {X 0,Y 552.97,Z 232.562,A -85,B 0,C 180,E1 25660.383,E2 25660.383} C_VEL
LIN {X 0,Y 559.369,Z 246.072,A -85,B 0,C 180,E1 25658.947,E2 25658.947} C_VEL
LIN {X 0,Y 560.441,Z 248.97,A -85,B 0,C 180,E1 25658.672,E2 25658.672} C_VEL
LIN {X 0,Y 558.666,Z 302.857,A -85,B 0,C 180,E1 25655.341,E2 25655.341} C_VEL
LIN {X 0,Y 557.1,Z 357.532,A -85,B 0,C 180,E1 25652.058,E2 25652.058} C_VEL
LIN {X 0,Y 555.679,Z 417.293,A -85,B 0,C 180,E1 25648.551,E2 25648.551} C_VEL
LIN {X 0,Y 556.397,Z 426.256,A -85,B 0,C 180,E1 25648.376,E2 25648.376} C_VEL
LIN {X 0,Y 555.439,Z 628.337,A -85,B 0,C 180,E1 25645.61,E2 25645.61} C_VEL
LIN {X 0,Y 555.169,Z 647.313,A -85,B 0,C 180,E1 25645.155,E2 25645.155} C_VEL
LIN {X 0,Y 554.833,Z 665.584,A -85,B 0,C 180,E1 25644.52,E2 25644.52} C_VEL
LIN {X 0,Y 554.435,Z 682.693,A -85,B 0,C 180,E1 25643.737,E2 25643.737} C_VEL
LIN {X 0,Y 553.999,Z 699.848,A -85,B 0,C 180,E1 25642.743,E2 25642.743} C_VEL
LIN {X 0,Y 553.564,Z 716.008,A -85,B 0,C 180,E1 25641.588,E2 25641.588} C_VEL
LIN {X 0,Y 553.147,Z 731.198,A -85,B 0,C 180,E1 25640.271,E2 25640.271} C_VEL
LIN {X 0,Y 552.787,Z 744.911,A -85,B 0,C 180,E1 25638.842,E2 25638.842} C_VEL
LIN {X 0,Y 552.483,Z 757.662,A -85,B 0,C 180,E1 25637.246,E2 25637.246} C_VEL
LIN {X 0,Y 552.246,Z 768.962,A -85,B 0,C 180,E1 25635.532,E2 25635.532} C_VEL
LIN {X 0,Y 552.094,Z 778.263,A -85,B 0,C 180,E1 25633.807,E2 25633.807} C_VEL
LIN {X 0,Y 551.987,Z 786.237,A -85,B 0,C 180,E1 25631.957,E2 25631.957} C_VEL
LIN {X 0,Y 551.941,Z 792.445,A -85,B 0,C 180,E1 25630.08,E2 25630.08} C_VEL
LIN {X 0,Y 551.914,Z 796.906,A -85,B 0,C 180,E1 25628.201,E2 25628.201} C_VEL
LIN {X 0,Y 551.917,Z 799.741,A -85,B 0,C 180,E1 25626.287,E2 25626.287} C_VEL
LIN {X 0,Y 551.912,Z 800.922,A -85,B 0,C 180,E1 25624.345,E2 25624.345} C_VEL
LIN {X 0,Y 551.912,Z 800.39,A -85,B 0,C 180,E1 25622.359,E2 25622.359} C_VEL
LIN {X 0,Y 551.914,Z 798.139,A -85,B 0,C 180,E1 25620.408,E2 25620.408} C_VEL
LIN {X 0,Y 551.93,Z 794.36,A -85,B 0,C 180,E1 25618.553,E2 25618.553} C_VEL
LIN {X 0,Y 551.964,Z 788.662,A -85,B 0,C 180,E1 25616.623,E2 25616.623} C_VEL
LIN {X 0,Y 552.051,Z 781.356,A -85,B 0,C 180,E1 25614.768,E2 25614.768} C_VEL
LIN {X 0,Y 552.185,Z 772.483,A -85,B 0,C 180,E1 25612.989,E2 25612.989} C_VEL
LIN {X 0,Y 552.389,Z 761.94,A -85,B 0,C 180,E1 25611.272,E2 25611.272} C_VEL
LIN {X 0,Y 552.667,Z 749.744,A -85,B 0,C 180,E1 25609.635,E2 25609.635} C_VEL
LIN {X 0,Y 553.012,Z 736.423,A -85,B 0,C 180,E1 25608.15,E2 25608.15} C_VEL
LIN {X 0,Y 553.408,Z 721.748,A -85,B 0,C 180,E1 25606.786,E2 25606.786} C_VEL
LIN {X 0,Y 553.853,Z 705.456,A -85,B 0,C 180,E1 25605.539,E2 25605.539} C_VEL
LIN {X 0,Y 554.268,Z 689.18,A -85,B 0,C 180,E1 25604.521,E2 25604.521} C_VEL
LIN {X 0,Y 554.698,Z 671.218,A -85,B 0,C 180,E1 25603.626,E2 25603.626} C_VEL
LIN {X 0,Y 555.069,Z 652.911,A -85,B 0,C 180,E1 25602.929,E2 25602.929} C_VEL
LIN {X 0,Y 555.357,Z 634.354,A -85,B 0,C 180,E1 25602.425,E2 25602.425} C_VEL
LIN {X 0,Y 555.545,Z 613.373,A -85,B 0,C 180,E1 25602.072,E2 25602.072} C_VEL
LIN {X 0,Y 556.281,Z 422.539,A -85,B 0,C 180,E1 25599.472,E2 25599.472} C_VEL
LIN {X 0,Y 555.667,Z 416.225,A -85,B 0,C 180,E1 25599.299,E2 25599.299} C_VEL
LIN {X 0,Y 557.189,Z 360.995,A -85,B 0,C 180,E1 25596.018,E2 25596.018} C_VEL
LIN {X 0,Y 559.056,Z 304.992,A -85,B 0,C 180,E1 25592.612,E2 25592.612} C_VEL
LIN {X 0,Y 561.098,Z 251.766,A -85,B 0,C 180,E1 25589.284,E2 25589.284} C_VEL
LIN {X 0,Y 561.054,Z 249.241,A -85,B 0,C 180,E1 25589.111,E2 25589.111} C_VEL
LIN {X 0,Y 553.316,Z 233.21,A -85,B 0,C 180,E1 25587.321,E2 25587.321} C_VEL
LIN {X 0,Y 552.351,Z 230.529,A -85,B 0,C 180,E1 25586.993,E2 25586.993} C_VEL
LIN {X 0,Y 552.286,Z 230.254,A -85,B 0,C 180,E1 25585.637,E2 25585.637} C_VEL
LIN {X 0,Y 552.262,Z 230.252,A -85,B 0,C 180,E1 25582.313,E2 25582.313} C_VEL
LIN {X 0,Y 552.311,Z 230.252,A -85,B 0,C 180,E1 25579.236,E2 25579.236} C_VEL
LIN {X 0,Y 552.258,Z 230.253,A -85,B 0,C 180,E1 25575.973,E2 25575.973} C_VEL
LIN {X 0,Y 552.33,Z 230.249,A -85,B 0,C 180,E1 25572.865,E2 25572.865} C_VEL
LIN {X 0,Y 552.256,Z 230.25,A -85,B 0,C 180,E1 25569.693,E2 25569.693} C_VEL
LIN {X 0,Y 552.31,Z 230.251,A -85,B 0,C 180,E1 25566.444,E2 25566.444} C_VEL
LIN {X 0,Y 552.26,Z 230.252,A -85,B 0,C 180,E1 25563.321,E2 25563.321} C_VEL
LIN {X 0,Y 552.269,Z 230.249,A -85,B 0,C 180,E1 25559.896,E2 25559.896} C_VEL
LIN {X 0,Y 552.278,Z 230.251,A -85,B 0,C 180,E1 25556.886,E2 25556.886} C_VEL
LIN {X 0,Y 552.259,Z 230.25,A -85,B 0,C 180,E1 25553.555,E2 25553.555} C_VEL
LIN {X 0,Y 552.298,Z 230.249,A -85,B 0,C 180,E1 25550.517,E2 25550.517} C_VEL
LIN {X 0,Y 552.254,Z 230.251,A -85,B 0,C 180,E1 25547.239,E2 25547.239} C_VEL
LIN {X 0,Y 552.33,Z 230.249,A -85,B 0,C 180,E1 25544.028,E2 25544.028} C_VEL
LIN {X 0,Y 552.254,Z 230.252,A -85,B 0,C 180,E1 25540.87,E2 25540.87} C_VEL
LIN {X 0,Y 552.306,Z 230.249,A -85,B 0,C 180,E1 25537.656,E2 25537.656} C_VEL
LIN {X 0,Y 552.259,Z 230.251,A -85,B 0,C 180,E1 25534.59,E2 25534.59} C_VEL
LIN {X 0,Y 552.289,Z 230.253,A -85,B 0,C 180,E1 25531.331,E2 25531.331} C_VEL
LIN {X 0,Y 552.265,Z 230.253,A -85,B 0,C 180,E1 25528.309,E2 25528.309} C_VEL
LIN {X 0,Y 552.264,Z 230.254,A -85,B 0,C 180,E1 25524.849,E2 25524.849} C_VEL
LIN {X 0,Y 552.3,Z 230.252,A -85,B 0,C 180,E1 25521.747,E2 25521.747} C_VEL
LIN {X 0,Y 552.259,Z 230.254,A -85,B 0,C 180,E1 25518.499,E2 25518.499} C_VEL
LIN {X 0,Y 552.288,Z 230.468,A -85,B 0,C 180,E1 25516.21,E2 25516.21} C_VEL
